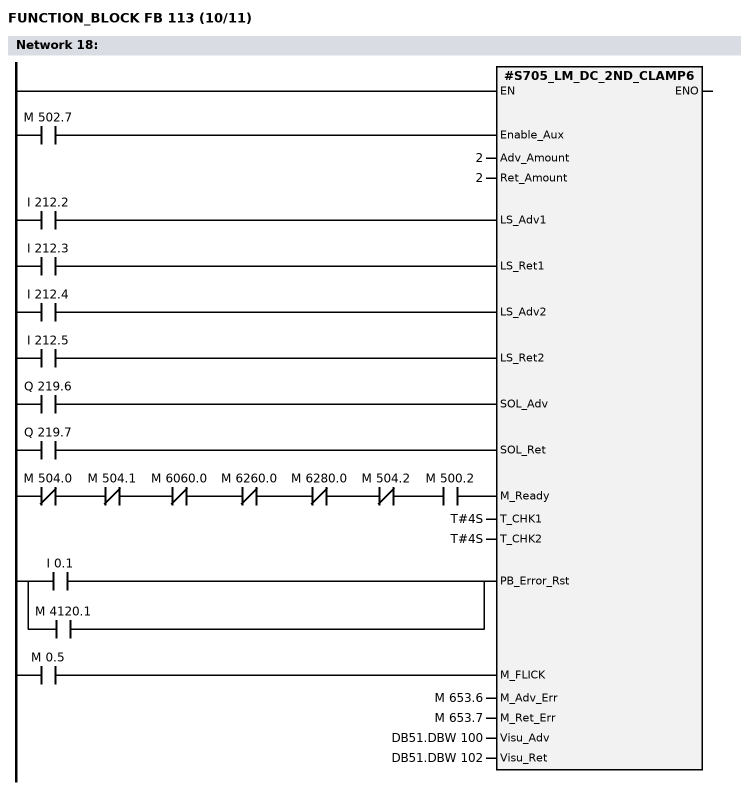

      A     M    502.7;
      =     L      0.0;
      BLD   103;
      A     I    212.2;
      =     L      0.1;
      BLD   103;
      A     I    212.3;
      =     L      0.2;
      BLD   103;
      A     I    212.4;
      =     L      0.3;
      BLD   103;
      A     I    212.5;
      =     L      0.4;
      BLD   103;
      A     Q    219.6;
      =     L      1.1;
      BLD   103;
      A     Q    219.7;
      =     L      1.2;
      BLD   103;
      AN    M    504.0;
      AN    M    504.1;
      AN    M   6060.0;
      AN    M   6260.0;
      AN    M   6280.0;
      AN    M    504.2;
      A     M    500.2;
      =     L      1.3;
      BLD   103;
      A(    ;
      O     I      0.1;
      O     M   4120.1;
      )     ;
      =     L      1.5;
      BLD   103;
      A     M      0.5;
      =     L      1.6;
      BLD   103;
      CALL #S705_LM_DC_2ND_CLAMP6 (
           Enable_Aux               := L      0.0,
           Adv_Amount               := 2,
           Ret_Amount               := 2,
           LS_Adv1                  := L      0.1,
           LS_Ret1                  := L      0.2,
           LS_Adv2                  := L      0.3,
           LS_Ret2                  := L      0.4,
           SOL_Adv                  := L      1.1,
           SOL_Ret                  := L      1.2,
           M_Ready                  := L      1.3,
           T_CHK1                   := T#4S,
           T_CHK2                   := T#4S,
           PB_Error_Rst             := L      1.5,
           M_FLICK                  := L      1.6,
           M_Adv_Err                := M    653.6,
           M_Ret_Err                := M    653.7,
           Visu_Adv                 := DB51.DBW  100,
           Visu_Ret                 := DB51.DBW  102);
      NOP   0;
NETWORK
TITLE =
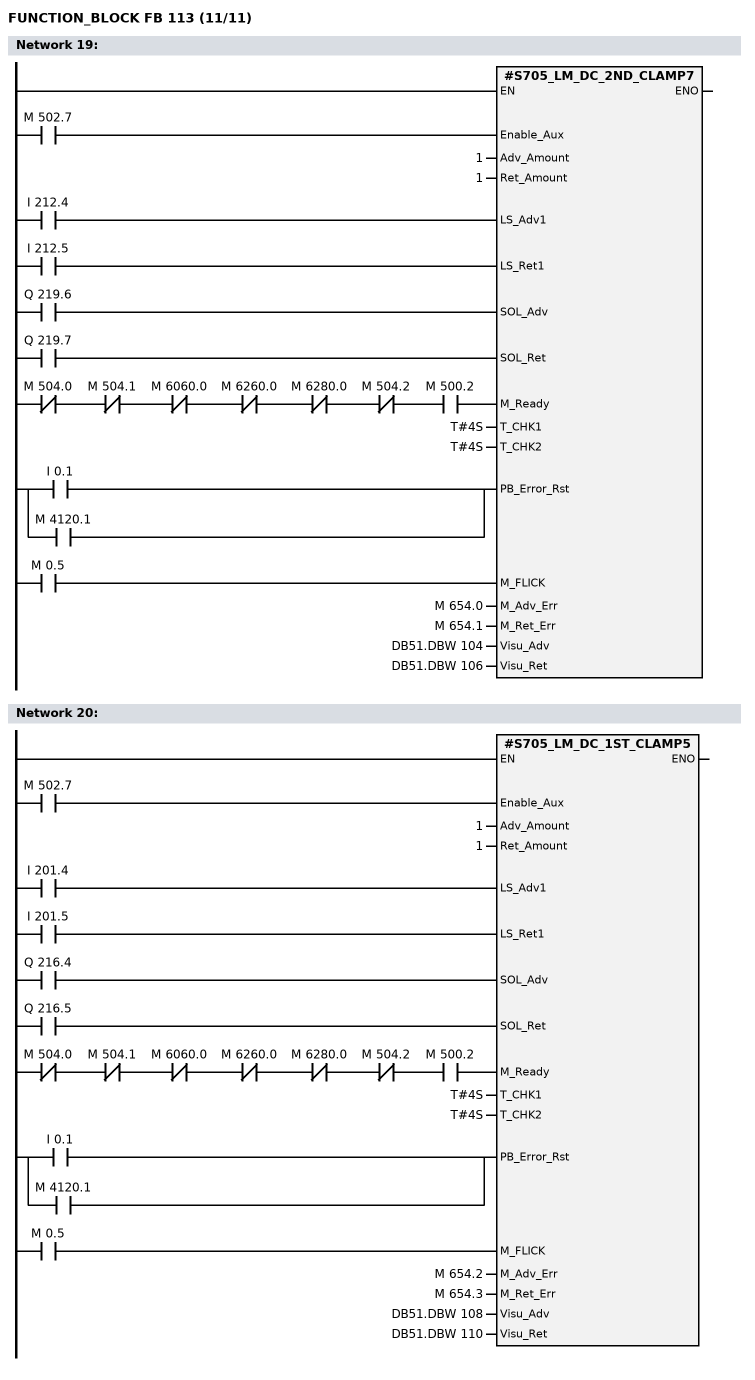

      A     M    502.7;
      =     L      0.0;
      BLD   103;
      A     I    212.4;
      =     L      0.1;
      BLD   103;
      A     I    212.5;
      =     L      0.2;
      BLD   103;
      A     Q    219.6;
      =     L      1.1;
      BLD   103;
      A     Q    219.7;
      =     L      1.2;
      BLD   103;
      AN    M    504.0;
      AN    M    504.1;
      AN    M   6060.0;
      AN    M   6260.0;
      AN    M   6280.0;
      AN    M    504.2;
      A     M    500.2;
      =     L      1.3;
      BLD   103;
      A(    ;
      O     I      0.1;
      O     M   4120.1;
      )     ;
      =     L      1.5;
      BLD   103;
      A     M      0.5;
      =     L      1.6;
      BLD   103;
      CALL #S705_LM_DC_2ND_CLAMP7 (
           Enable_Aux               := L      0.0,
           Adv_Amount               := 1,
           Ret_Amount               := 1,
           LS_Adv1                  := L      0.1,
           LS_Ret1                  := L      0.2,
           SOL_Adv                  := L      1.1,
           SOL_Ret                  := L      1.2,
           M_Ready                  := L      1.3,
           T_CHK1                   := T#4S,
           T_CHK2                   := T#4S,
           PB_Error_Rst             := L      1.5,
           M_FLICK                  := L      1.6,
           M_Adv_Err                := M    654.0,
           M_Ret_Err                := M    654.1,
           Visu_Adv                 := DB51.DBW  104,
           Visu_Ret                 := DB51.DBW  106);
      NOP   0;
NETWORK
TITLE =

      A     M    502.7;
      =     L      0.0;
      BLD   103;
      A     I    201.4;
      =     L      0.1;
      BLD   103;
      A     I    201.5;
      =     L      0.2;
      BLD   103;
      A     Q    216.4;
      =     L      1.1;
      BLD   103;
      A     Q    216.5;
      =     L      1.2;
      BLD   103;
      AN    M    504.0;
      AN    M    504.1;
      AN    M   6060.0;
      AN    M   6260.0;
      AN    M   6280.0;
      AN    M    504.2;
      A     M    500.2;
      =     L      1.3;
      BLD   103;
      A(    ;
      O     I      0.1;
      O     M   4120.1;
      )     ;
      =     L      1.5;
      BLD   103;
      A     M      0.5;
      =     L      1.6;
      BLD   103;
      CALL #S705_LM_DC_1ST_CLAMP5 (
           Enable_Aux               := L      0.0,
           Adv_Amount               := 1,
           Ret_Amount               := 1,
           LS_Adv1                  := L      0.1,
           LS_Ret1                  := L      0.2,
           SOL_Adv                  := L      1.1,
           SOL_Ret                  := L      1.2,
           M_Ready                  := L      1.3,
           T_CHK1                   := T#4S,
           T_CHK2                   := T#4S,
           PB_Error_Rst             := L      1.5,
           M_FLICK                  := L      1.6,
           M_Adv_Err                := M    654.2,
           M_Ret_Err                := M    654.3,
           Visu_Adv                 := DB51.DBW  108,
           Visu_Ret                 := DB51.DBW  110);
      NOP   0;
END_FUNCTION_BLOCK

DATA_BLOCK DB 113
TITLE =
VERSION : 0.0

 FB 113
BEGIN
   S705_LM_DC_PIN.Enable_Aux := FALSE;
   S705_LM_DC_PIN.Adv_Amount := 1;
   S705_LM_DC_PIN.Ret_Amount := 1;
   S705_LM_DC_PIN.LS_Adv1 := FALSE;
   S705_LM_DC_PIN.LS_Ret1 := FALSE;
   S705_LM_DC_PIN.LS_Adv2 := FALSE;
   S705_LM_DC_PIN.LS_Ret2 := FALSE;
   S705_LM_DC_PIN.LS_Adv3 := FALSE;
   S705_LM_DC_PIN.LS_Ret3 := FALSE;
   S705_LM_DC_PIN.LS_Adv4 := FALSE;
   S705_LM_DC_PIN.LS_Ret4 := FALSE;
   S705_LM_DC_PIN.SOL_Adv := FALSE;
   S705_LM_DC_PIN.SOL_Ret := FALSE;
   S705_LM_DC_PIN.M_Ready := TRUE;
   S705_LM_DC_PIN.T_CHK1 := T#4S;
   S705_LM_DC_PIN.T_CHK2 := T#4S;
   S705_LM_DC_PIN.PB_Lamp_CHK := FALSE;
   S705_LM_DC_PIN.PB_Error_Rst := FALSE;
   S705_LM_DC_PIN.M_FLICK := TRUE;
   S705_LM_DC_PIN.M_Adv_Err := FALSE;
   S705_LM_DC_PIN.M_Ret_Err := FALSE;
   S705_LM_DC_PIN.LP_Adv := FALSE;
   S705_LM_DC_PIN.LP_Ret := FALSE;
   S705_LM_DC_PIN.Visu_Adv := W#16#0;
   S705_LM_DC_PIN.Visu_Ret := W#16#0;
   S705_LM_DC_PIN.Error_T1.IN := FALSE;
   S705_LM_DC_PIN.Error_T1.PT := T#4S;
   S705_LM_DC_PIN.Error_T1.Q := FALSE;
   S705_LM_DC_PIN.Error_T1.ET := T#0MS;
   S705_LM_DC_PIN.Error_T1.STATE := B#16#0;
   S705_LM_DC_PIN.Error_T1.STIME := T#15D15H9M7S743MS;
   S705_LM_DC_PIN.Error_T1.ATIME := T#15D15H9M7S788MS;
   S705_LM_DC_PIN.Error_T2.IN := FALSE;
   S705_LM_DC_PIN.Error_T2.PT := T#4S;
   S705_LM_DC_PIN.Error_T2.Q := FALSE;
   S705_LM_DC_PIN.Error_T2.ET := T#0MS;
   S705_LM_DC_PIN.Error_T2.STATE := B#16#0;
   S705_LM_DC_PIN.Error_T2.STIME := T#0MS;
   S705_LM_DC_PIN.Error_T2.ATIME := T#0MS;
   S705_LM_DC_PIN.CHK_Aux1 := FALSE;
   S705_LM_DC_PIN.CHK_Aux2 := FALSE;
   S705_LM_DC_PIN.Error_T1_DN := FALSE;
   S705_LM_DC_PIN.Error_T2_DN := FALSE;
   S705_LM_DC_PIN.Adv_Memo := TRUE;
   S705_LM_DC_PIN.Visu_Adv_Arr[0] := FALSE;
   S705_LM_DC_PIN.Visu_Adv_Arr[1] := FALSE;
   S705_LM_DC_PIN.Visu_Adv_Arr[2] := FALSE;
   S705_LM_DC_PIN.Visu_Adv_Arr[3] := FALSE;
   S705_LM_DC_PIN.Visu_Adv_Arr[4] := FALSE;
   S705_LM_DC_PIN.Visu_Adv_Arr[5] := FALSE;
   S705_LM_DC_PIN.Visu_Adv_Arr[6] := FALSE;
   S705_LM_DC_PIN.Visu_Adv_Arr[7] := FALSE;
   S705_LM_DC_PIN.Visu_Adv_Arr[8] := FALSE;
   S705_LM_DC_PIN.Visu_Adv_Arr[9] := FALSE;
   S705_LM_DC_PIN.Visu_Adv_Arr[10] := FALSE;
   S705_LM_DC_PIN.Visu_Adv_Arr[11] := FALSE;
   S705_LM_DC_PIN.Visu_Adv_Arr[12] := FALSE;
   S705_LM_DC_PIN.Visu_Adv_Arr[13] := FALSE;
   S705_LM_DC_PIN.Visu_Adv_Arr[14] := FALSE;
   S705_LM_DC_PIN.Visu_Adv_Arr[15] := FALSE;
   S705_LM_DC_PIN.Visu_Ret_Arr[0] := FALSE;
   S705_LM_DC_PIN.Visu_Ret_Arr[1] := FALSE;
   S705_LM_DC_PIN.Visu_Ret_Arr[2] := FALSE;
   S705_LM_DC_PIN.Visu_Ret_Arr[3] := FALSE;
   S705_LM_DC_PIN.Visu_Ret_Arr[4] := FALSE;
   S705_LM_DC_PIN.Visu_Ret_Arr[5] := FALSE;
   S705_LM_DC_PIN.Visu_Ret_Arr[6] := FALSE;
   S705_LM_DC_PIN.Visu_Ret_Arr[7] := FALSE;
   S705_LM_DC_PIN.Visu_Ret_Arr[8] := FALSE;
   S705_LM_DC_PIN.Visu_Ret_Arr[9] := FALSE;
   S705_LM_DC_PIN.Visu_Ret_Arr[10] := FALSE;
   S705_LM_DC_PIN.Visu_Ret_Arr[11] := FALSE;
   S705_LM_DC_PIN.Visu_Ret_Arr[12] := FALSE;
   S705_LM_DC_PIN.Visu_Ret_Arr[13] := FALSE;
   S705_LM_DC_PIN.Visu_Ret_Arr[14] := FALSE;
   S705_LM_DC_PIN.Visu_Ret_Arr[15] := FALSE;
   S705_LM_DC_PIN.BLK_Move_Ret := 0;
   S705_LM_DC_PIN.Enable := FALSE;
   S705_LM_DC_PIN.Adv_End := FALSE;
   S705_LM_DC_PIN.Ret_End := FALSE;
   S705_LM_DC_1ST_CLAMP1.Enable_Aux := FALSE;
   S705_LM_DC_1ST_CLAMP1.Adv_Amount := 1;
   S705_LM_DC_1ST_CLAMP1.Ret_Amount := 1;
   S705_LM_DC_1ST_CLAMP1.LS_Adv1 := FALSE;
   S705_LM_DC_1ST_CLAMP1.LS_Ret1 := FALSE;
   S705_LM_DC_1ST_CLAMP1.LS_Adv2 := FALSE;
   S705_LM_DC_1ST_CLAMP1.LS_Ret2 := FALSE;
   S705_LM_DC_1ST_CLAMP1.LS_Adv3 := FALSE;
   S705_LM_DC_1ST_CLAMP1.LS_Ret3 := FALSE;
   S705_LM_DC_1ST_CLAMP1.LS_Adv4 := FALSE;
   S705_LM_DC_1ST_CLAMP1.LS_Ret4 := FALSE;
   S705_LM_DC_1ST_CLAMP1.SOL_Adv := FALSE;
   S705_LM_DC_1ST_CLAMP1.SOL_Ret := FALSE;
   S705_LM_DC_1ST_CLAMP1.M_Ready := TRUE;
   S705_LM_DC_1ST_CLAMP1.T_CHK1 := T#4S;
   S705_LM_DC_1ST_CLAMP1.T_CHK2 := T#4S;
   S705_LM_DC_1ST_CLAMP1.PB_Lamp_CHK := FALSE;
   S705_LM_DC_1ST_CLAMP1.PB_Error_Rst := FALSE;
   S705_LM_DC_1ST_CLAMP1.M_FLICK := TRUE;
   S705_LM_DC_1ST_CLAMP1.M_Adv_Err := FALSE;
   S705_LM_DC_1ST_CLAMP1.M_Ret_Err := FALSE;
   S705_LM_DC_1ST_CLAMP1.LP_Adv := FALSE;
   S705_LM_DC_1ST_CLAMP1.LP_Ret := FALSE;
   S705_LM_DC_1ST_CLAMP1.Visu_Adv := W#16#0;
   S705_LM_DC_1ST_CLAMP1.Visu_Ret := W#16#0;
   S705_LM_DC_1ST_CLAMP1.Error_T1.IN := FALSE;
   S705_LM_DC_1ST_CLAMP1.Error_T1.PT := T#4S;
   S705_LM_DC_1ST_CLAMP1.Error_T1.Q := FALSE;
   S705_LM_DC_1ST_CLAMP1.Error_T1.ET := T#0MS;
   S705_LM_DC_1ST_CLAMP1.Error_T1.STATE := B#16#0;
   S705_LM_DC_1ST_CLAMP1.Error_T1.STIME := T#15D15H9M7S743MS;
   S705_LM_DC_1ST_CLAMP1.Error_T1.ATIME := T#15D15H9M7S788MS;
   S705_LM_DC_1ST_CLAMP1.Error_T2.IN := FALSE;
   S705_LM_DC_1ST_CLAMP1.Error_T2.PT := T#4S;
   S705_LM_DC_1ST_CLAMP1.Error_T2.Q := FALSE;
   S705_LM_DC_1ST_CLAMP1.Error_T2.ET := T#0MS;
   S705_LM_DC_1ST_CLAMP1.Error_T2.STATE := B#16#0;
   S705_LM_DC_1ST_CLAMP1.Error_T2.STIME := T#0MS;
   S705_LM_DC_1ST_CLAMP1.Error_T2.ATIME := T#0MS;
   S705_LM_DC_1ST_CLAMP1.CHK_Aux1 := FALSE;
   S705_LM_DC_1ST_CLAMP1.CHK_Aux2 := FALSE;
   S705_LM_DC_1ST_CLAMP1.Error_T1_DN := FALSE;
   S705_LM_DC_1ST_CLAMP1.Error_T2_DN := FALSE;
   S705_LM_DC_1ST_CLAMP1.Adv_Memo := TRUE;
   S705_LM_DC_1ST_CLAMP1.Visu_Adv_Arr[0] := FALSE;
   S705_LM_DC_1ST_CLAMP1.Visu_Adv_Arr[1] := FALSE;
   S705_LM_DC_1ST_CLAMP1.Visu_Adv_Arr[2] := FALSE;
   S705_LM_DC_1ST_CLAMP1.Visu_Adv_Arr[3] := FALSE;
   S705_LM_DC_1ST_CLAMP1.Visu_Adv_Arr[4] := FALSE;
   S705_LM_DC_1ST_CLAMP1.Visu_Adv_Arr[5] := FALSE;
   S705_LM_DC_1ST_CLAMP1.Visu_Adv_Arr[6] := FALSE;
   S705_LM_DC_1ST_CLAMP1.Visu_Adv_Arr[7] := FALSE;
   S705_LM_DC_1ST_CLAMP1.Visu_Adv_Arr[8] := FALSE;
   S705_LM_DC_1ST_CLAMP1.Visu_Adv_Arr[9] := FALSE;
   S705_LM_DC_1ST_CLAMP1.Visu_Adv_Arr[10] := FALSE;
   S705_LM_DC_1ST_CLAMP1.Visu_Adv_Arr[11] := FALSE;
   S705_LM_DC_1ST_CLAMP1.Visu_Adv_Arr[12] := FALSE;
   S705_LM_DC_1ST_CLAMP1.Visu_Adv_Arr[13] := FALSE;
   S705_LM_DC_1ST_CLAMP1.Visu_Adv_Arr[14] := FALSE;
   S705_LM_DC_1ST_CLAMP1.Visu_Adv_Arr[15] := FALSE;
   S705_LM_DC_1ST_CLAMP1.Visu_Ret_Arr[0] := FALSE;
   S705_LM_DC_1ST_CLAMP1.Visu_Ret_Arr[1] := FALSE;
   S705_LM_DC_1ST_CLAMP1.Visu_Ret_Arr[2] := FALSE;
   S705_LM_DC_1ST_CLAMP1.Visu_Ret_Arr[3] := FALSE;
   S705_LM_DC_1ST_CLAMP1.Visu_Ret_Arr[4] := FALSE;
   S705_LM_DC_1ST_CLAMP1.Visu_Ret_Arr[5] := FALSE;
   S705_LM_DC_1ST_CLAMP1.Visu_Ret_Arr[6] := FALSE;
   S705_LM_DC_1ST_CLAMP1.Visu_Ret_Arr[7] := FALSE;
   S705_LM_DC_1ST_CLAMP1.Visu_Ret_Arr[8] := FALSE;
   S705_LM_DC_1ST_CLAMP1.Visu_Ret_Arr[9] := FALSE;
   S705_LM_DC_1ST_CLAMP1.Visu_Ret_Arr[10] := FALSE;
   S705_LM_DC_1ST_CLAMP1.Visu_Ret_Arr[11] := FALSE;
   S705_LM_DC_1ST_CLAMP1.Visu_Ret_Arr[12] := FALSE;
   S705_LM_DC_1ST_CLAMP1.Visu_Ret_Arr[13] := FALSE;
   S705_LM_DC_1ST_CLAMP1.Visu_Ret_Arr[14] := FALSE;
   S705_LM_DC_1ST_CLAMP1.Visu_Ret_Arr[15] := FALSE;
   S705_LM_DC_1ST_CLAMP1.BLK_Move_Ret := 0;
   S705_LM_DC_1ST_CLAMP1.Enable := FALSE;
   S705_LM_DC_1ST_CLAMP1.Adv_End := FALSE;
   S705_LM_DC_1ST_CLAMP1.Ret_End := FALSE;
   S705_LM_DC_1ST_CLAMP2.Enable_Aux := FALSE;
   S705_LM_DC_1ST_CLAMP2.Adv_Amount := 2;
   S705_LM_DC_1ST_CLAMP2.Ret_Amount := 2;
   S705_LM_DC_1ST_CLAMP2.LS_Adv1 := FALSE;
   S705_LM_DC_1ST_CLAMP2.LS_Ret1 := FALSE;
   S705_LM_DC_1ST_CLAMP2.LS_Adv2 := FALSE;
   S705_LM_DC_1ST_CLAMP2.LS_Ret2 := FALSE;
   S705_LM_DC_1ST_CLAMP2.LS_Adv3 := FALSE;
   S705_LM_DC_1ST_CLAMP2.LS_Ret3 := FALSE;
   S705_LM_DC_1ST_CLAMP2.LS_Adv4 := FALSE;
   S705_LM_DC_1ST_CLAMP2.LS_Ret4 := FALSE;
   S705_LM_DC_1ST_CLAMP2.SOL_Adv := FALSE;
   S705_LM_DC_1ST_CLAMP2.SOL_Ret := FALSE;
   S705_LM_DC_1ST_CLAMP2.M_Ready := TRUE;
   S705_LM_DC_1ST_CLAMP2.T_CHK1 := T#4S;
   S705_LM_DC_1ST_CLAMP2.T_CHK2 := T#4S;
   S705_LM_DC_1ST_CLAMP2.PB_Lamp_CHK := FALSE;
   S705_LM_DC_1ST_CLAMP2.PB_Error_Rst := FALSE;
   S705_LM_DC_1ST_CLAMP2.M_FLICK := TRUE;
   S705_LM_DC_1ST_CLAMP2.M_Adv_Err := FALSE;
   S705_LM_DC_1ST_CLAMP2.M_Ret_Err := FALSE;
   S705_LM_DC_1ST_CLAMP2.LP_Adv := FALSE;
   S705_LM_DC_1ST_CLAMP2.LP_Ret := FALSE;
   S705_LM_DC_1ST_CLAMP2.Visu_Adv := W#16#0;
   S705_LM_DC_1ST_CLAMP2.Visu_Ret := W#16#0;
   S705_LM_DC_1ST_CLAMP2.Error_T1.IN := FALSE;
   S705_LM_DC_1ST_CLAMP2.Error_T1.PT := T#4S;
   S705_LM_DC_1ST_CLAMP2.Error_T1.Q := FALSE;
   S705_LM_DC_1ST_CLAMP2.Error_T1.ET := T#0MS;
   S705_LM_DC_1ST_CLAMP2.Error_T1.STATE := B#16#0;
   S705_LM_DC_1ST_CLAMP2.Error_T1.STIME := T#22D22H55M12S68MS;
   S705_LM_DC_1ST_CLAMP2.Error_T1.ATIME := T#22D22H55M12S817MS;
   S705_LM_DC_1ST_CLAMP2.Error_T2.IN := FALSE;
   S705_LM_DC_1ST_CLAMP2.Error_T2.PT := T#4S;
   S705_LM_DC_1ST_CLAMP2.Error_T2.Q := FALSE;
   S705_LM_DC_1ST_CLAMP2.Error_T2.ET := T#0MS;
   S705_LM_DC_1ST_CLAMP2.Error_T2.STATE := B#16#0;
   S705_LM_DC_1ST_CLAMP2.Error_T2.STIME := T#0MS;
   S705_LM_DC_1ST_CLAMP2.Error_T2.ATIME := T#0MS;
   S705_LM_DC_1ST_CLAMP2.CHK_Aux1 := FALSE;
   S705_LM_DC_1ST_CLAMP2.CHK_Aux2 := FALSE;
   S705_LM_DC_1ST_CLAMP2.Error_T1_DN := FALSE;
   S705_LM_DC_1ST_CLAMP2.Error_T2_DN := FALSE;
   S705_LM_DC_1ST_CLAMP2.Adv_Memo := TRUE;
   S705_LM_DC_1ST_CLAMP2.Visu_Adv_Arr[0] := FALSE;
   S705_LM_DC_1ST_CLAMP2.Visu_Adv_Arr[1] := FALSE;
   S705_LM_DC_1ST_CLAMP2.Visu_Adv_Arr[2] := FALSE;
   S705_LM_DC_1ST_CLAMP2.Visu_Adv_Arr[3] := FALSE;
   S705_LM_DC_1ST_CLAMP2.Visu_Adv_Arr[4] := FALSE;
   S705_LM_DC_1ST_CLAMP2.Visu_Adv_Arr[5] := FALSE;
   S705_LM_DC_1ST_CLAMP2.Visu_Adv_Arr[6] := FALSE;
   S705_LM_DC_1ST_CLAMP2.Visu_Adv_Arr[7] := FALSE;
   S705_LM_DC_1ST_CLAMP2.Visu_Adv_Arr[8] := FALSE;
   S705_LM_DC_1ST_CLAMP2.Visu_Adv_Arr[9] := FALSE;
   S705_LM_DC_1ST_CLAMP2.Visu_Adv_Arr[10] := FALSE;
   S705_LM_DC_1ST_CLAMP2.Visu_Adv_Arr[11] := FALSE;
   S705_LM_DC_1ST_CLAMP2.Visu_Adv_Arr[12] := FALSE;
   S705_LM_DC_1ST_CLAMP2.Visu_Adv_Arr[13] := FALSE;
   S705_LM_DC_1ST_CLAMP2.Visu_Adv_Arr[14] := FALSE;
   S705_LM_DC_1ST_CLAMP2.Visu_Adv_Arr[15] := FALSE;
   S705_LM_DC_1ST_CLAMP2.Visu_Ret_Arr[0] := FALSE;
   S705_LM_DC_1ST_CLAMP2.Visu_Ret_Arr[1] := FALSE;
   S705_LM_DC_1ST_CLAMP2.Visu_Ret_Arr[2] := FALSE;
   S705_LM_DC_1ST_CLAMP2.Visu_Ret_Arr[3] := FALSE;
   S705_LM_DC_1ST_CLAMP2.Visu_Ret_Arr[4] := FALSE;
   S705_LM_DC_1ST_CLAMP2.Visu_Ret_Arr[5] := FALSE;
   S705_LM_DC_1ST_CLAMP2.Visu_Ret_Arr[6] := FALSE;
   S705_LM_DC_1ST_CLAMP2.Visu_Ret_Arr[7] := FALSE;
   S705_LM_DC_1ST_CLAMP2.Visu_Ret_Arr[8] := FALSE;
   S705_LM_DC_1ST_CLAMP2.Visu_Ret_Arr[9] := FALSE;
   S705_LM_DC_1ST_CLAMP2.Visu_Ret_Arr[10] := FALSE;
   S705_LM_DC_1ST_CLAMP2.Visu_Ret_Arr[11] := FALSE;
   S705_LM_DC_1ST_CLAMP2.Visu_Ret_Arr[12] := FALSE;
   S705_LM_DC_1ST_CLAMP2.Visu_Ret_Arr[13] := FALSE;
   S705_LM_DC_1ST_CLAMP2.Visu_Ret_Arr[14] := FALSE;
   S705_LM_DC_1ST_CLAMP2.Visu_Ret_Arr[15] := FALSE;
   S705_LM_DC_1ST_CLAMP2.BLK_Move_Ret := 0;
   S705_LM_DC_1ST_CLAMP2.Enable := FALSE;
   S705_LM_DC_1ST_CLAMP2.Adv_End := FALSE;
   S705_LM_DC_1ST_CLAMP2.Ret_End := FALSE;
   S705_LM_DC_1ST_CLAMP3.Enable_Aux := FALSE;
   S705_LM_DC_1ST_CLAMP3.Adv_Amount := 1;
   S705_LM_DC_1ST_CLAMP3.Ret_Amount := 1;
   S705_LM_DC_1ST_CLAMP3.LS_Adv1 := FALSE;
   S705_LM_DC_1ST_CLAMP3.LS_Ret1 := FALSE;
   S705_LM_DC_1ST_CLAMP3.LS_Adv2 := FALSE;
   S705_LM_DC_1ST_CLAMP3.LS_Ret2 := FALSE;
   S705_LM_DC_1ST_CLAMP3.LS_Adv3 := FALSE;
   S705_LM_DC_1ST_CLAMP3.LS_Ret3 := FALSE;
   S705_LM_DC_1ST_CLAMP3.LS_Adv4 := FALSE;
   S705_LM_DC_1ST_CLAMP3.LS_Ret4 := FALSE;
   S705_LM_DC_1ST_CLAMP3.SOL_Adv := FALSE;
   S705_LM_DC_1ST_CLAMP3.SOL_Ret := FALSE;
   S705_LM_DC_1ST_CLAMP3.M_Ready := TRUE;
   S705_LM_DC_1ST_CLAMP3.T_CHK1 := T#4S;
   S705_LM_DC_1ST_CLAMP3.T_CHK2 := T#4S;
   S705_LM_DC_1ST_CLAMP3.PB_Lamp_CHK := FALSE;
   S705_LM_DC_1ST_CLAMP3.PB_Error_Rst := FALSE;
   S705_LM_DC_1ST_CLAMP3.M_FLICK := TRUE;
   S705_LM_DC_1ST_CLAMP3.M_Adv_Err := FALSE;
   S705_LM_DC_1ST_CLAMP3.M_Ret_Err := FALSE;
   S705_LM_DC_1ST_CLAMP3.LP_Adv := FALSE;
   S705_LM_DC_1ST_CLAMP3.LP_Ret := FALSE;
   S705_LM_DC_1ST_CLAMP3.Visu_Adv := W#16#0;
   S705_LM_DC_1ST_CLAMP3.Visu_Ret := W#16#0;
   S705_LM_DC_1ST_CLAMP3.Error_T1.IN := FALSE;
   S705_LM_DC_1ST_CLAMP3.Error_T1.PT := T#4S;
   S705_LM_DC_1ST_CLAMP3.Error_T1.Q := FALSE;
   S705_LM_DC_1ST_CLAMP3.Error_T1.ET := T#0MS;
   S705_LM_DC_1ST_CLAMP3.Error_T1.STATE := B#16#0;
   S705_LM_DC_1ST_CLAMP3.Error_T1.STIME := T#22D22H55M12S68MS;
   S705_LM_DC_1ST_CLAMP3.Error_T1.ATIME := T#22D22H55M12S726MS;
   S705_LM_DC_1ST_CLAMP3.Error_T2.IN := FALSE;
   S705_LM_DC_1ST_CLAMP3.Error_T2.PT := T#4S;
   S705_LM_DC_1ST_CLAMP3.Error_T2.Q := FALSE;
   S705_LM_DC_1ST_CLAMP3.Error_T2.ET := T#0MS;
   S705_LM_DC_1ST_CLAMP3.Error_T2.STATE := B#16#0;
   S705_LM_DC_1ST_CLAMP3.Error_T2.STIME := T#0MS;
   S705_LM_DC_1ST_CLAMP3.Error_T2.ATIME := T#0MS;
   S705_LM_DC_1ST_CLAMP3.CHK_Aux1 := FALSE;
   S705_LM_DC_1ST_CLAMP3.CHK_Aux2 := FALSE;
   S705_LM_DC_1ST_CLAMP3.Error_T1_DN := FALSE;
   S705_LM_DC_1ST_CLAMP3.Error_T2_DN := FALSE;
   S705_LM_DC_1ST_CLAMP3.Adv_Memo := TRUE;
   S705_LM_DC_1ST_CLAMP3.Visu_Adv_Arr[0] := FALSE;
   S705_LM_DC_1ST_CLAMP3.Visu_Adv_Arr[1] := FALSE;
   S705_LM_DC_1ST_CLAMP3.Visu_Adv_Arr[2] := FALSE;
   S705_LM_DC_1ST_CLAMP3.Visu_Adv_Arr[3] := FALSE;
   S705_LM_DC_1ST_CLAMP3.Visu_Adv_Arr[4] := FALSE;
   S705_LM_DC_1ST_CLAMP3.Visu_Adv_Arr[5] := FALSE;
   S705_LM_DC_1ST_CLAMP3.Visu_Adv_Arr[6] := FALSE;
   S705_LM_DC_1ST_CLAMP3.Visu_Adv_Arr[7] := FALSE;
   S705_LM_DC_1ST_CLAMP3.Visu_Adv_Arr[8] := FALSE;
   S705_LM_DC_1ST_CLAMP3.Visu_Adv_Arr[9] := FALSE;
   S705_LM_DC_1ST_CLAMP3.Visu_Adv_Arr[10] := FALSE;
   S705_LM_DC_1ST_CLAMP3.Visu_Adv_Arr[11] := FALSE;
   S705_LM_DC_1ST_CLAMP3.Visu_Adv_Arr[12] := FALSE;
   S705_LM_DC_1ST_CLAMP3.Visu_Adv_Arr[13] := FALSE;
   S705_LM_DC_1ST_CLAMP3.Visu_Adv_Arr[14] := FALSE;
   S705_LM_DC_1ST_CLAMP3.Visu_Adv_Arr[15] := FALSE;
   S705_LM_DC_1ST_CLAMP3.Visu_Ret_Arr[0] := FALSE;
   S705_LM_DC_1ST_CLAMP3.Visu_Ret_Arr[1] := FALSE;
   S705_LM_DC_1ST_CLAMP3.Visu_Ret_Arr[2] := FALSE;
   S705_LM_DC_1ST_CLAMP3.Visu_Ret_Arr[3] := FALSE;
   S705_LM_DC_1ST_CLAMP3.Visu_Ret_Arr[4] := FALSE;
   S705_LM_DC_1ST_CLAMP3.Visu_Ret_Arr[5] := FALSE;
   S705_LM_DC_1ST_CLAMP3.Visu_Ret_Arr[6] := FALSE;
   S705_LM_DC_1ST_CLAMP3.Visu_Ret_Arr[7] := FALSE;
   S705_LM_DC_1ST_CLAMP3.Visu_Ret_Arr[8] := FALSE;
   S705_LM_DC_1ST_CLAMP3.Visu_Ret_Arr[9] := FALSE;
   S705_LM_DC_1ST_CLAMP3.Visu_Ret_Arr[10] := FALSE;
   S705_LM_DC_1ST_CLAMP3.Visu_Ret_Arr[11] := FALSE;
   S705_LM_DC_1ST_CLAMP3.Visu_Ret_Arr[12] := FALSE;
   S705_LM_DC_1ST_CLAMP3.Visu_Ret_Arr[13] := FALSE;
   S705_LM_DC_1ST_CLAMP3.Visu_Ret_Arr[14] := FALSE;
   S705_LM_DC_1ST_CLAMP3.Visu_Ret_Arr[15] := FALSE;
   S705_LM_DC_1ST_CLAMP3.BLK_Move_Ret := 0;
   S705_LM_DC_1ST_CLAMP3.Enable := FALSE;
   S705_LM_DC_1ST_CLAMP3.Adv_End := FALSE;
   S705_LM_DC_1ST_CLAMP3.Ret_End := FALSE;
   S705_LM_DC_1ST_CLAMP4.Enable_Aux := FALSE;
   S705_LM_DC_1ST_CLAMP4.Adv_Amount := 1;
   S705_LM_DC_1ST_CLAMP4.Ret_Amount := 1;
   S705_LM_DC_1ST_CLAMP4.LS_Adv1 := FALSE;
   S705_LM_DC_1ST_CLAMP4.LS_Ret1 := FALSE;
   S705_LM_DC_1ST_CLAMP4.LS_Adv2 := FALSE;
   S705_LM_DC_1ST_CLAMP4.LS_Ret2 := FALSE;
   S705_LM_DC_1ST_CLAMP4.LS_Adv3 := FALSE;
   S705_LM_DC_1ST_CLAMP4.LS_Ret3 := FALSE;
   S705_LM_DC_1ST_CLAMP4.LS_Adv4 := FALSE;
   S705_LM_DC_1ST_CLAMP4.LS_Ret4 := FALSE;
   S705_LM_DC_1ST_CLAMP4.SOL_Adv := FALSE;
   S705_LM_DC_1ST_CLAMP4.SOL_Ret := FALSE;
   S705_LM_DC_1ST_CLAMP4.M_Ready := TRUE;
   S705_LM_DC_1ST_CLAMP4.T_CHK1 := T#4S;
   S705_LM_DC_1ST_CLAMP4.T_CHK2 := T#4S;
   S705_LM_DC_1ST_CLAMP4.PB_Lamp_CHK := FALSE;
   S705_LM_DC_1ST_CLAMP4.PB_Error_Rst := FALSE;
   S705_LM_DC_1ST_CLAMP4.M_FLICK := TRUE;
   S705_LM_DC_1ST_CLAMP4.M_Adv_Err := FALSE;
   S705_LM_DC_1ST_CLAMP4.M_Ret_Err := FALSE;
   S705_LM_DC_1ST_CLAMP4.LP_Adv := FALSE;
   S705_LM_DC_1ST_CLAMP4.LP_Ret := FALSE;
   S705_LM_DC_1ST_CLAMP4.Visu_Adv := W#16#0;
   S705_LM_DC_1ST_CLAMP4.Visu_Ret := W#16#0;
   S705_LM_DC_1ST_CLAMP4.Error_T1.IN := FALSE;
   S705_LM_DC_1ST_CLAMP4.Error_T1.PT := T#4S;
   S705_LM_DC_1ST_CLAMP4.Error_T1.Q := FALSE;
   S705_LM_DC_1ST_CLAMP4.Error_T1.ET := T#0MS;
   S705_LM_DC_1ST_CLAMP4.Error_T1.STATE := B#16#0;
   S705_LM_DC_1ST_CLAMP4.Error_T1.STIME := T#22D22H55M13S;
   S705_LM_DC_1ST_CLAMP4.Error_T1.ATIME := T#22D22H55M13S46MS;
   S705_LM_DC_1ST_CLAMP4.Error_T2.IN := FALSE;
   S705_LM_DC_1ST_CLAMP4.Error_T2.PT := T#4S;
   S705_LM_DC_1ST_CLAMP4.Error_T2.Q := FALSE;
   S705_LM_DC_1ST_CLAMP4.Error_T2.ET := T#0MS;
   S705_LM_DC_1ST_CLAMP4.Error_T2.STATE := B#16#0;
   S705_LM_DC_1ST_CLAMP4.Error_T2.STIME := T#0MS;
   S705_LM_DC_1ST_CLAMP4.Error_T2.ATIME := T#0MS;
   S705_LM_DC_1ST_CLAMP4.CHK_Aux1 := FALSE;
   S705_LM_DC_1ST_CLAMP4.CHK_Aux2 := FALSE;
   S705_LM_DC_1ST_CLAMP4.Error_T1_DN := FALSE;
   S705_LM_DC_1ST_CLAMP4.Error_T2_DN := FALSE;
   S705_LM_DC_1ST_CLAMP4.Adv_Memo := TRUE;
   S705_LM_DC_1ST_CLAMP4.Visu_Adv_Arr[0] := FALSE;
   S705_LM_DC_1ST_CLAMP4.Visu_Adv_Arr[1] := FALSE;
   S705_LM_DC_1ST_CLAMP4.Visu_Adv_Arr[2] := FALSE;
   S705_LM_DC_1ST_CLAMP4.Visu_Adv_Arr[3] := FALSE;
   S705_LM_DC_1ST_CLAMP4.Visu_Adv_Arr[4] := FALSE;
   S705_LM_DC_1ST_CLAMP4.Visu_Adv_Arr[5] := FALSE;
   S705_LM_DC_1ST_CLAMP4.Visu_Adv_Arr[6] := FALSE;
   S705_LM_DC_1ST_CLAMP4.Visu_Adv_Arr[7] := FALSE;
   S705_LM_DC_1ST_CLAMP4.Visu_Adv_Arr[8] := FALSE;
   S705_LM_DC_1ST_CLAMP4.Visu_Adv_Arr[9] := FALSE;
   S705_LM_DC_1ST_CLAMP4.Visu_Adv_Arr[10] := FALSE;
   S705_LM_DC_1ST_CLAMP4.Visu_Adv_Arr[11] := FALSE;
   S705_LM_DC_1ST_CLAMP4.Visu_Adv_Arr[12] := FALSE;
   S705_LM_DC_1ST_CLAMP4.Visu_Adv_Arr[13] := FALSE;
   S705_LM_DC_1ST_CLAMP4.Visu_Adv_Arr[14] := FALSE;
   S705_LM_DC_1ST_CLAMP4.Visu_Adv_Arr[15] := FALSE;
   S705_LM_DC_1ST_CLAMP4.Visu_Ret_Arr[0] := FALSE;
   S705_LM_DC_1ST_CLAMP4.Visu_Ret_Arr[1] := FALSE;
   S705_LM_DC_1ST_CLAMP4.Visu_Ret_Arr[2] := FALSE;
   S705_LM_DC_1ST_CLAMP4.Visu_Ret_Arr[3] := FALSE;
   S705_LM_DC_1ST_CLAMP4.Visu_Ret_Arr[4] := FALSE;
   S705_LM_DC_1ST_CLAMP4.Visu_Ret_Arr[5] := FALSE;
   S705_LM_DC_1ST_CLAMP4.Visu_Ret_Arr[6] := FALSE;
   S705_LM_DC_1ST_CLAMP4.Visu_Ret_Arr[7] := FALSE;
   S705_LM_DC_1ST_CLAMP4.Visu_Ret_Arr[8] := FALSE;
   S705_LM_DC_1ST_CLAMP4.Visu_Ret_Arr[9] := FALSE;
   S705_LM_DC_1ST_CLAMP4.Visu_Ret_Arr[10] := FALSE;
   S705_LM_DC_1ST_CLAMP4.Visu_Ret_Arr[11] := FALSE;
   S705_LM_DC_1ST_CLAMP4.Visu_Ret_Arr[12] := FALSE;
   S705_LM_DC_1ST_CLAMP4.Visu_Ret_Arr[13] := FALSE;
   S705_LM_DC_1ST_CLAMP4.Visu_Ret_Arr[14] := FALSE;
   S705_LM_DC_1ST_CLAMP4.Visu_Ret_Arr[15] := FALSE;
   S705_LM_DC_1ST_CLAMP4.BLK_Move_Ret := 0;
   S705_LM_DC_1ST_CLAMP4.Enable := FALSE;
   S705_LM_DC_1ST_CLAMP4.Adv_End := FALSE;
   S705_LM_DC_1ST_CLAMP4.Ret_End := FALSE;
   S705_LM_DC_2ND_CLAMP1.Enable_Aux := FALSE;
   S705_LM_DC_2ND_CLAMP1.Adv_Amount := 2;
   S705_LM_DC_2ND_CLAMP1.Ret_Amount := 1;
   S705_LM_DC_2ND_CLAMP1.LS_Adv1 := FALSE;
   S705_LM_DC_2ND_CLAMP1.LS_Ret1 := FALSE;
   S705_LM_DC_2ND_CLAMP1.LS_Adv2 := FALSE;
   S705_LM_DC_2ND_CLAMP1.LS_Ret2 := FALSE;
   S705_LM_DC_2ND_CLAMP1.LS_Adv3 := FALSE;
   S705_LM_DC_2ND_CLAMP1.LS_Ret3 := FALSE;
   S705_LM_DC_2ND_CLAMP1.LS_Adv4 := FALSE;
   S705_LM_DC_2ND_CLAMP1.LS_Ret4 := FALSE;
   S705_LM_DC_2ND_CLAMP1.SOL_Adv := FALSE;
   S705_LM_DC_2ND_CLAMP1.SOL_Ret := FALSE;
   S705_LM_DC_2ND_CLAMP1.M_Ready := TRUE;
   S705_LM_DC_2ND_CLAMP1.T_CHK1 := T#4S;
   S705_LM_DC_2ND_CLAMP1.T_CHK2 := T#4S;
   S705_LM_DC_2ND_CLAMP1.PB_Lamp_CHK := FALSE;
   S705_LM_DC_2ND_CLAMP1.PB_Error_Rst := FALSE;
   S705_LM_DC_2ND_CLAMP1.M_FLICK := TRUE;
   S705_LM_DC_2ND_CLAMP1.M_Adv_Err := FALSE;
   S705_LM_DC_2ND_CLAMP1.M_Ret_Err := FALSE;
   S705_LM_DC_2ND_CLAMP1.LP_Adv := FALSE;
   S705_LM_DC_2ND_CLAMP1.LP_Ret := FALSE;
   S705_LM_DC_2ND_CLAMP1.Visu_Adv := W#16#0;
   S705_LM_DC_2ND_CLAMP1.Visu_Ret := W#16#0;
   S705_LM_DC_2ND_CLAMP1.Error_T1.IN := FALSE;
   S705_LM_DC_2ND_CLAMP1.Error_T1.PT := T#4S;
   S705_LM_DC_2ND_CLAMP1.Error_T1.Q := FALSE;
   S705_LM_DC_2ND_CLAMP1.Error_T1.ET := T#0MS;
   S705_LM_DC_2ND_CLAMP1.Error_T1.STATE := B#16#0;
   S705_LM_DC_2ND_CLAMP1.Error_T1.STIME := T#22D22H55M35S537MS;
   S705_LM_DC_2ND_CLAMP1.Error_T1.ATIME := T#22D22H55M36S828MS;
   S705_LM_DC_2ND_CLAMP1.Error_T2.IN := FALSE;
   S705_LM_DC_2ND_CLAMP1.Error_T2.PT := T#4S;
   S705_LM_DC_2ND_CLAMP1.Error_T2.Q := FALSE;
   S705_LM_DC_2ND_CLAMP1.Error_T2.ET := T#0MS;
   S705_LM_DC_2ND_CLAMP1.Error_T2.STATE := B#16#0;
   S705_LM_DC_2ND_CLAMP1.Error_T2.STIME := T#0MS;
   S705_LM_DC_2ND_CLAMP1.Error_T2.ATIME := T#0MS;
   S705_LM_DC_2ND_CLAMP1.CHK_Aux1 := FALSE;
   S705_LM_DC_2ND_CLAMP1.CHK_Aux2 := FALSE;
   S705_LM_DC_2ND_CLAMP1.Error_T1_DN := FALSE;
   S705_LM_DC_2ND_CLAMP1.Error_T2_DN := FALSE;
   S705_LM_DC_2ND_CLAMP1.Adv_Memo := TRUE;
   S705_LM_DC_2ND_CLAMP1.Visu_Adv_Arr[0] := FALSE;
   S705_LM_DC_2ND_CLAMP1.Visu_Adv_Arr[1] := FALSE;
   S705_LM_DC_2ND_CLAMP1.Visu_Adv_Arr[2] := FALSE;
   S705_LM_DC_2ND_CLAMP1.Visu_Adv_Arr[3] := FALSE;
   S705_LM_DC_2ND_CLAMP1.Visu_Adv_Arr[4] := FALSE;
   S705_LM_DC_2ND_CLAMP1.Visu_Adv_Arr[5] := FALSE;
   S705_LM_DC_2ND_CLAMP1.Visu_Adv_Arr[6] := FALSE;
   S705_LM_DC_2ND_CLAMP1.Visu_Adv_Arr[7] := FALSE;
   S705_LM_DC_2ND_CLAMP1.Visu_Adv_Arr[8] := FALSE;
   S705_LM_DC_2ND_CLAMP1.Visu_Adv_Arr[9] := FALSE;
   S705_LM_DC_2ND_CLAMP1.Visu_Adv_Arr[10] := FALSE;
   S705_LM_DC_2ND_CLAMP1.Visu_Adv_Arr[11] := FALSE;
   S705_LM_DC_2ND_CLAMP1.Visu_Adv_Arr[12] := FALSE;
   S705_LM_DC_2ND_CLAMP1.Visu_Adv_Arr[13] := FALSE;
   S705_LM_DC_2ND_CLAMP1.Visu_Adv_Arr[14] := FALSE;
   S705_LM_DC_2ND_CLAMP1.Visu_Adv_Arr[15] := FALSE;
   S705_LM_DC_2ND_CLAMP1.Visu_Ret_Arr[0] := FALSE;
   S705_LM_DC_2ND_CLAMP1.Visu_Ret_Arr[1] := FALSE;
   S705_LM_DC_2ND_CLAMP1.Visu_Ret_Arr[2] := FALSE;
   S705_LM_DC_2ND_CLAMP1.Visu_Ret_Arr[3] := FALSE;
   S705_LM_DC_2ND_CLAMP1.Visu_Ret_Arr[4] := FALSE;
   S705_LM_DC_2ND_CLAMP1.Visu_Ret_Arr[5] := FALSE;
   S705_LM_DC_2ND_CLAMP1.Visu_Ret_Arr[6] := FALSE;
   S705_LM_DC_2ND_CLAMP1.Visu_Ret_Arr[7] := FALSE;
   S705_LM_DC_2ND_CLAMP1.Visu_Ret_Arr[8] := FALSE;
   S705_LM_DC_2ND_CLAMP1.Visu_Ret_Arr[9] := FALSE;
   S705_LM_DC_2ND_CLAMP1.Visu_Ret_Arr[10] := FALSE;
   S705_LM_DC_2ND_CLAMP1.Visu_Ret_Arr[11] := FALSE;
   S705_LM_DC_2ND_CLAMP1.Visu_Ret_Arr[12] := FALSE;
   S705_LM_DC_2ND_CLAMP1.Visu_Ret_Arr[13] := FALSE;
   S705_LM_DC_2ND_CLAMP1.Visu_Ret_Arr[14] := FALSE;
   S705_LM_DC_2ND_CLAMP1.Visu_Ret_Arr[15] := FALSE;
   S705_LM_DC_2ND_CLAMP1.BLK_Move_Ret := 0;
   S705_LM_DC_2ND_CLAMP1.Enable := FALSE;
   S705_LM_DC_2ND_CLAMP1.Adv_End := FALSE;
   S705_LM_DC_2ND_CLAMP1.Ret_End := FALSE;
   S705_LM_DC_2ND_CLAMP2.Enable_Aux := FALSE;
   S705_LM_DC_2ND_CLAMP2.Adv_Amount := 1;
   S705_LM_DC_2ND_CLAMP2.Ret_Amount := 1;
   S705_LM_DC_2ND_CLAMP2.LS_Adv1 := FALSE;
   S705_LM_DC_2ND_CLAMP2.LS_Ret1 := FALSE;
   S705_LM_DC_2ND_CLAMP2.LS_Adv2 := FALSE;
   S705_LM_DC_2ND_CLAMP2.LS_Ret2 := FALSE;
   S705_LM_DC_2ND_CLAMP2.LS_Adv3 := FALSE;
   S705_LM_DC_2ND_CLAMP2.LS_Ret3 := FALSE;
   S705_LM_DC_2ND_CLAMP2.LS_Adv4 := FALSE;
   S705_LM_DC_2ND_CLAMP2.LS_Ret4 := FALSE;
   S705_LM_DC_2ND_CLAMP2.SOL_Adv := FALSE;
   S705_LM_DC_2ND_CLAMP2.SOL_Ret := FALSE;
   S705_LM_DC_2ND_CLAMP2.M_Ready := TRUE;
   S705_LM_DC_2ND_CLAMP2.T_CHK1 := T#4S;
   S705_LM_DC_2ND_CLAMP2.T_CHK2 := T#4S;
   S705_LM_DC_2ND_CLAMP2.PB_Lamp_CHK := FALSE;
   S705_LM_DC_2ND_CLAMP2.PB_Error_Rst := FALSE;
   S705_LM_DC_2ND_CLAMP2.M_FLICK := TRUE;
   S705_LM_DC_2ND_CLAMP2.M_Adv_Err := FALSE;
   S705_LM_DC_2ND_CLAMP2.M_Ret_Err := FALSE;
   S705_LM_DC_2ND_CLAMP2.LP_Adv := FALSE;
   S705_LM_DC_2ND_CLAMP2.LP_Ret := FALSE;
   S705_LM_DC_2ND_CLAMP2.Visu_Adv := W#16#0;
   S705_LM_DC_2ND_CLAMP2.Visu_Ret := W#16#0;
   S705_LM_DC_2ND_CLAMP2.Error_T1.IN := FALSE;
   S705_LM_DC_2ND_CLAMP2.Error_T1.PT := T#4S;
   S705_LM_DC_2ND_CLAMP2.Error_T1.Q := FALSE;
   S705_LM_DC_2ND_CLAMP2.Error_T1.ET := T#0MS;
   S705_LM_DC_2ND_CLAMP2.Error_T1.STATE := B#16#0;
   S705_LM_DC_2ND_CLAMP2.Error_T1.STIME := T#22D22H55M12S68MS;
   S705_LM_DC_2ND_CLAMP2.Error_T1.ATIME := T#22D22H55M13S364MS;
   S705_LM_DC_2ND_CLAMP2.Error_T2.IN := FALSE;
   S705_LM_DC_2ND_CLAMP2.Error_T2.PT := T#4S;
   S705_LM_DC_2ND_CLAMP2.Error_T2.Q := FALSE;
   S705_LM_DC_2ND_CLAMP2.Error_T2.ET := T#0MS;
   S705_LM_DC_2ND_CLAMP2.Error_T2.STATE := B#16#0;
   S705_LM_DC_2ND_CLAMP2.Error_T2.STIME := T#0MS;
   S705_LM_DC_2ND_CLAMP2.Error_T2.ATIME := T#0MS;
   S705_LM_DC_2ND_CLAMP2.CHK_Aux1 := FALSE;
   S705_LM_DC_2ND_CLAMP2.CHK_Aux2 := FALSE;
   S705_LM_DC_2ND_CLAMP2.Error_T1_DN := FALSE;
   S705_LM_DC_2ND_CLAMP2.Error_T2_DN := FALSE;
   S705_LM_DC_2ND_CLAMP2.Adv_Memo := TRUE;
   S705_LM_DC_2ND_CLAMP2.Visu_Adv_Arr[0] := FALSE;
   S705_LM_DC_2ND_CLAMP2.Visu_Adv_Arr[1] := FALSE;
   S705_LM_DC_2ND_CLAMP2.Visu_Adv_Arr[2] := FALSE;
   S705_LM_DC_2ND_CLAMP2.Visu_Adv_Arr[3] := FALSE;
   S705_LM_DC_2ND_CLAMP2.Visu_Adv_Arr[4] := FALSE;
   S705_LM_DC_2ND_CLAMP2.Visu_Adv_Arr[5] := FALSE;
   S705_LM_DC_2ND_CLAMP2.Visu_Adv_Arr[6] := FALSE;
   S705_LM_DC_2ND_CLAMP2.Visu_Adv_Arr[7] := FALSE;
   S705_LM_DC_2ND_CLAMP2.Visu_Adv_Arr[8] := FALSE;
   S705_LM_DC_2ND_CLAMP2.Visu_Adv_Arr[9] := FALSE;
   S705_LM_DC_2ND_CLAMP2.Visu_Adv_Arr[10] := FALSE;
   S705_LM_DC_2ND_CLAMP2.Visu_Adv_Arr[11] := FALSE;
   S705_LM_DC_2ND_CLAMP2.Visu_Adv_Arr[12] := FALSE;
   S705_LM_DC_2ND_CLAMP2.Visu_Adv_Arr[13] := FALSE;
   S705_LM_DC_2ND_CLAMP2.Visu_Adv_Arr[14] := FALSE;
   S705_LM_DC_2ND_CLAMP2.Visu_Adv_Arr[15] := FALSE;
   S705_LM_DC_2ND_CLAMP2.Visu_Ret_Arr[0] := FALSE;
   S705_LM_DC_2ND_CLAMP2.Visu_Ret_Arr[1] := FALSE;
   S705_LM_DC_2ND_CLAMP2.Visu_Ret_Arr[2] := FALSE;
   S705_LM_DC_2ND_CLAMP2.Visu_Ret_Arr[3] := FALSE;
   S705_LM_DC_2ND_CLAMP2.Visu_Ret_Arr[4] := FALSE;
   S705_LM_DC_2ND_CLAMP2.Visu_Ret_Arr[5] := FALSE;
   S705_LM_DC_2ND_CLAMP2.Visu_Ret_Arr[6] := FALSE;
   S705_LM_DC_2ND_CLAMP2.Visu_Ret_Arr[7] := FALSE;
   S705_LM_DC_2ND_CLAMP2.Visu_Ret_Arr[8] := FALSE;
   S705_LM_DC_2ND_CLAMP2.Visu_Ret_Arr[9] := FALSE;
   S705_LM_DC_2ND_CLAMP2.Visu_Ret_Arr[10] := FALSE;
   S705_LM_DC_2ND_CLAMP2.Visu_Ret_Arr[11] := FALSE;
   S705_LM_DC_2ND_CLAMP2.Visu_Ret_Arr[12] := FALSE;
   S705_LM_DC_2ND_CLAMP2.Visu_Ret_Arr[13] := FALSE;
   S705_LM_DC_2ND_CLAMP2.Visu_Ret_Arr[14] := FALSE;
   S705_LM_DC_2ND_CLAMP2.Visu_Ret_Arr[15] := FALSE;
   S705_LM_DC_2ND_CLAMP2.BLK_Move_Ret := 0;
   S705_LM_DC_2ND_CLAMP2.Enable := FALSE;
   S705_LM_DC_2ND_CLAMP2.Adv_End := FALSE;
   S705_LM_DC_2ND_CLAMP2.Ret_End := FALSE;
   S705_LM_DC_2ND_CLAMP3.Enable_Aux := FALSE;
   S705_LM_DC_2ND_CLAMP3.Adv_Amount := 1;
   S705_LM_DC_2ND_CLAMP3.Ret_Amount := 1;
   S705_LM_DC_2ND_CLAMP3.LS_Adv1 := FALSE;
   S705_LM_DC_2ND_CLAMP3.LS_Ret1 := FALSE;
   S705_LM_DC_2ND_CLAMP3.LS_Adv2 := FALSE;
   S705_LM_DC_2ND_CLAMP3.LS_Ret2 := FALSE;
   S705_LM_DC_2ND_CLAMP3.LS_Adv3 := FALSE;
   S705_LM_DC_2ND_CLAMP3.LS_Ret3 := FALSE;
   S705_LM_DC_2ND_CLAMP3.LS_Adv4 := FALSE;
   S705_LM_DC_2ND_CLAMP3.LS_Ret4 := FALSE;
   S705_LM_DC_2ND_CLAMP3.SOL_Adv := FALSE;
   S705_LM_DC_2ND_CLAMP3.SOL_Ret := FALSE;
   S705_LM_DC_2ND_CLAMP3.M_Ready := TRUE;
   S705_LM_DC_2ND_CLAMP3.T_CHK1 := T#4S;
   S705_LM_DC_2ND_CLAMP3.T_CHK2 := T#4S;
   S705_LM_DC_2ND_CLAMP3.PB_Lamp_CHK := FALSE;
   S705_LM_DC_2ND_CLAMP3.PB_Error_Rst := FALSE;
   S705_LM_DC_2ND_CLAMP3.M_FLICK := TRUE;
   S705_LM_DC_2ND_CLAMP3.M_Adv_Err := FALSE;
   S705_LM_DC_2ND_CLAMP3.M_Ret_Err := FALSE;
   S705_LM_DC_2ND_CLAMP3.LP_Adv := FALSE;
   S705_LM_DC_2ND_CLAMP3.LP_Ret := FALSE;
   S705_LM_DC_2ND_CLAMP3.Visu_Adv := W#16#0;
   S705_LM_DC_2ND_CLAMP3.Visu_Ret := W#16#0;
   S705_LM_DC_2ND_CLAMP3.Error_T1.IN := FALSE;
   S705_LM_DC_2ND_CLAMP3.Error_T1.PT := T#4S;
   S705_LM_DC_2ND_CLAMP3.Error_T1.Q := FALSE;
   S705_LM_DC_2ND_CLAMP3.Error_T1.ET := T#0MS;
   S705_LM_DC_2ND_CLAMP3.Error_T1.STATE := B#16#0;
   S705_LM_DC_2ND_CLAMP3.Error_T1.STIME := T#22D22H55M13S364MS;
   S705_LM_DC_2ND_CLAMP3.Error_T1.ATIME := T#22D22H55M14S182MS;
   S705_LM_DC_2ND_CLAMP3.Error_T2.IN := FALSE;
   S705_LM_DC_2ND_CLAMP3.Error_T2.PT := T#4S;
   S705_LM_DC_2ND_CLAMP3.Error_T2.Q := FALSE;
   S705_LM_DC_2ND_CLAMP3.Error_T2.ET := T#0MS;
   S705_LM_DC_2ND_CLAMP3.Error_T2.STATE := B#16#0;
   S705_LM_DC_2ND_CLAMP3.Error_T2.STIME := T#0MS;
   S705_LM_DC_2ND_CLAMP3.Error_T2.ATIME := T#0MS;
   S705_LM_DC_2ND_CLAMP3.CHK_Aux1 := FALSE;
   S705_LM_DC_2ND_CLAMP3.CHK_Aux2 := FALSE;
   S705_LM_DC_2ND_CLAMP3.Error_T1_DN := FALSE;
   S705_LM_DC_2ND_CLAMP3.Error_T2_DN := FALSE;
   S705_LM_DC_2ND_CLAMP3.Adv_Memo := TRUE;
   S705_LM_DC_2ND_CLAMP3.Visu_Adv_Arr[0] := FALSE;
   S705_LM_DC_2ND_CLAMP3.Visu_Adv_Arr[1] := FALSE;
   S705_LM_DC_2ND_CLAMP3.Visu_Adv_Arr[2] := FALSE;
   S705_LM_DC_2ND_CLAMP3.Visu_Adv_Arr[3] := FALSE;
   S705_LM_DC_2ND_CLAMP3.Visu_Adv_Arr[4] := FALSE;
   S705_LM_DC_2ND_CLAMP3.Visu_Adv_Arr[5] := FALSE;
   S705_LM_DC_2ND_CLAMP3.Visu_Adv_Arr[6] := FALSE;
   S705_LM_DC_2ND_CLAMP3.Visu_Adv_Arr[7] := FALSE;
   S705_LM_DC_2ND_CLAMP3.Visu_Adv_Arr[8] := FALSE;
   S705_LM_DC_2ND_CLAMP3.Visu_Adv_Arr[9] := FALSE;
   S705_LM_DC_2ND_CLAMP3.Visu_Adv_Arr[10] := FALSE;
   S705_LM_DC_2ND_CLAMP3.Visu_Adv_Arr[11] := FALSE;
   S705_LM_DC_2ND_CLAMP3.Visu_Adv_Arr[12] := FALSE;
   S705_LM_DC_2ND_CLAMP3.Visu_Adv_Arr[13] := FALSE;
   S705_LM_DC_2ND_CLAMP3.Visu_Adv_Arr[14] := FALSE;
   S705_LM_DC_2ND_CLAMP3.Visu_Adv_Arr[15] := FALSE;
   S705_LM_DC_2ND_CLAMP3.Visu_Ret_Arr[0] := FALSE;
   S705_LM_DC_2ND_CLAMP3.Visu_Ret_Arr[1] := FALSE;
   S705_LM_DC_2ND_CLAMP3.Visu_Ret_Arr[2] := FALSE;
   S705_LM_DC_2ND_CLAMP3.Visu_Ret_Arr[3] := FALSE;
   S705_LM_DC_2ND_CLAMP3.Visu_Ret_Arr[4] := FALSE;
   S705_LM_DC_2ND_CLAMP3.Visu_Ret_Arr[5] := FALSE;
   S705_LM_DC_2ND_CLAMP3.Visu_Ret_Arr[6] := FALSE;
   S705_LM_DC_2ND_CLAMP3.Visu_Ret_Arr[7] := FALSE;
   S705_LM_DC_2ND_CLAMP3.Visu_Ret_Arr[8] := FALSE;
   S705_LM_DC_2ND_CLAMP3.Visu_Ret_Arr[9] := FALSE;
   S705_LM_DC_2ND_CLAMP3.Visu_Ret_Arr[10] := FALSE;
   S705_LM_DC_2ND_CLAMP3.Visu_Ret_Arr[11] := FALSE;
   S705_LM_DC_2ND_CLAMP3.Visu_Ret_Arr[12] := FALSE;
   S705_LM_DC_2ND_CLAMP3.Visu_Ret_Arr[13] := FALSE;
   S705_LM_DC_2ND_CLAMP3.Visu_Ret_Arr[14] := FALSE;
   S705_LM_DC_2ND_CLAMP3.Visu_Ret_Arr[15] := FALSE;
   S705_LM_DC_2ND_CLAMP3.BLK_Move_Ret := 0;
   S705_LM_DC_2ND_CLAMP3.Enable := FALSE;
   S705_LM_DC_2ND_CLAMP3.Adv_End := FALSE;
   S705_LM_DC_2ND_CLAMP3.Ret_End := FALSE;
   S705_LM_DC_2ND_CLAMP4.Enable_Aux := FALSE;
   S705_LM_DC_2ND_CLAMP4.Adv_Amount := 1;
   S705_LM_DC_2ND_CLAMP4.Ret_Amount := 1;
   S705_LM_DC_2ND_CLAMP4.LS_Adv1 := FALSE;
   S705_LM_DC_2ND_CLAMP4.LS_Ret1 := FALSE;
   S705_LM_DC_2ND_CLAMP4.LS_Adv2 := FALSE;
   S705_LM_DC_2ND_CLAMP4.LS_Ret2 := FALSE;
   S705_LM_DC_2ND_CLAMP4.LS_Adv3 := FALSE;
   S705_LM_DC_2ND_CLAMP4.LS_Ret3 := FALSE;
   S705_LM_DC_2ND_CLAMP4.LS_Adv4 := FALSE;
   S705_LM_DC_2ND_CLAMP4.LS_Ret4 := FALSE;
   S705_LM_DC_2ND_CLAMP4.SOL_Adv := FALSE;
   S705_LM_DC_2ND_CLAMP4.SOL_Ret := FALSE;
   S705_LM_DC_2ND_CLAMP4.M_Ready := TRUE;
   S705_LM_DC_2ND_CLAMP4.T_CHK1 := T#4S;
   S705_LM_DC_2ND_CLAMP4.T_CHK2 := T#4S;
   S705_LM_DC_2ND_CLAMP4.PB_Lamp_CHK := FALSE;
   S705_LM_DC_2ND_CLAMP4.PB_Error_Rst := FALSE;
   S705_LM_DC_2ND_CLAMP4.M_FLICK := TRUE;
   S705_LM_DC_2ND_CLAMP4.M_Adv_Err := FALSE;
   S705_LM_DC_2ND_CLAMP4.M_Ret_Err := FALSE;
   S705_LM_DC_2ND_CLAMP4.LP_Adv := FALSE;
   S705_LM_DC_2ND_CLAMP4.LP_Ret := FALSE;
   S705_LM_DC_2ND_CLAMP4.Visu_Adv := W#16#0;
   S705_LM_DC_2ND_CLAMP4.Visu_Ret := W#16#0;
   S705_LM_DC_2ND_CLAMP4.Error_T1.IN := FALSE;
   S705_LM_DC_2ND_CLAMP4.Error_T1.PT := T#4S;
   S705_LM_DC_2ND_CLAMP4.Error_T1.Q := FALSE;
   S705_LM_DC_2ND_CLAMP4.Error_T1.ET := T#0MS;
   S705_LM_DC_2ND_CLAMP4.Error_T1.STATE := B#16#0;
   S705_LM_DC_2ND_CLAMP4.Error_T1.STIME := T#22D22H55M12S726MS;
   S705_LM_DC_2ND_CLAMP4.Error_T1.ATIME := T#22D22H55M13S364MS;
   S705_LM_DC_2ND_CLAMP4.Error_T2.IN := FALSE;
   S705_LM_DC_2ND_CLAMP4.Error_T2.PT := T#4S;
   S705_LM_DC_2ND_CLAMP4.Error_T2.Q := FALSE;
   S705_LM_DC_2ND_CLAMP4.Error_T2.ET := T#0MS;
   S705_LM_DC_2ND_CLAMP4.Error_T2.STATE := B#16#0;
   S705_LM_DC_2ND_CLAMP4.Error_T2.STIME := T#0MS;
   S705_LM_DC_2ND_CLAMP4.Error_T2.ATIME := T#0MS;
   S705_LM_DC_2ND_CLAMP4.CHK_Aux1 := FALSE;
   S705_LM_DC_2ND_CLAMP4.CHK_Aux2 := FALSE;
   S705_LM_DC_2ND_CLAMP4.Error_T1_DN := FALSE;
   S705_LM_DC_2ND_CLAMP4.Error_T2_DN := FALSE;
   S705_LM_DC_2ND_CLAMP4.Adv_Memo := TRUE;
   S705_LM_DC_2ND_CLAMP4.Visu_Adv_Arr[0] := FALSE;
   S705_LM_DC_2ND_CLAMP4.Visu_Adv_Arr[1] := FALSE;
   S705_LM_DC_2ND_CLAMP4.Visu_Adv_Arr[2] := FALSE;
   S705_LM_DC_2ND_CLAMP4.Visu_Adv_Arr[3] := FALSE;
   S705_LM_DC_2ND_CLAMP4.Visu_Adv_Arr[4] := FALSE;
   S705_LM_DC_2ND_CLAMP4.Visu_Adv_Arr[5] := FALSE;
   S705_LM_DC_2ND_CLAMP4.Visu_Adv_Arr[6] := FALSE;
   S705_LM_DC_2ND_CLAMP4.Visu_Adv_Arr[7] := FALSE;
   S705_LM_DC_2ND_CLAMP4.Visu_Adv_Arr[8] := FALSE;
   S705_LM_DC_2ND_CLAMP4.Visu_Adv_Arr[9] := FALSE;
   S705_LM_DC_2ND_CLAMP4.Visu_Adv_Arr[10] := FALSE;
   S705_LM_DC_2ND_CLAMP4.Visu_Adv_Arr[11] := FALSE;
   S705_LM_DC_2ND_CLAMP4.Visu_Adv_Arr[12] := FALSE;
   S705_LM_DC_2ND_CLAMP4.Visu_Adv_Arr[13] := FALSE;
   S705_LM_DC_2ND_CLAMP4.Visu_Adv_Arr[14] := FALSE;
   S705_LM_DC_2ND_CLAMP4.Visu_Adv_Arr[15] := FALSE;
   S705_LM_DC_2ND_CLAMP4.Visu_Ret_Arr[0] := FALSE;
   S705_LM_DC_2ND_CLAMP4.Visu_Ret_Arr[1] := FALSE;
   S705_LM_DC_2ND_CLAMP4.Visu_Ret_Arr[2] := FALSE;
   S705_LM_DC_2ND_CLAMP4.Visu_Ret_Arr[3] := FALSE;
   S705_LM_DC_2ND_CLAMP4.Visu_Ret_Arr[4] := FALSE;
   S705_LM_DC_2ND_CLAMP4.Visu_Ret_Arr[5] := FALSE;
   S705_LM_DC_2ND_CLAMP4.Visu_Ret_Arr[6] := FALSE;
   S705_LM_DC_2ND_CLAMP4.Visu_Ret_Arr[7] := FALSE;
   S705_LM_DC_2ND_CLAMP4.Visu_Ret_Arr[8] := FALSE;
   S705_LM_DC_2ND_CLAMP4.Visu_Ret_Arr[9] := FALSE;
   S705_LM_DC_2ND_CLAMP4.Visu_Ret_Arr[10] := FALSE;
   S705_LM_DC_2ND_CLAMP4.Visu_Ret_Arr[11] := FALSE;
   S705_LM_DC_2ND_CLAMP4.Visu_Ret_Arr[12] := FALSE;
   S705_LM_DC_2ND_CLAMP4.Visu_Ret_Arr[13] := FALSE;
   S705_LM_DC_2ND_CLAMP4.Visu_Ret_Arr[14] := FALSE;
   S705_LM_DC_2ND_CLAMP4.Visu_Ret_Arr[15] := FALSE;
   S705_LM_DC_2ND_CLAMP4.BLK_Move_Ret := 0;
   S705_LM_DC_2ND_CLAMP4.Enable := FALSE;
   S705_LM_DC_2ND_CLAMP4.Adv_End := FALSE;
   S705_LM_DC_2ND_CLAMP4.Ret_End := FALSE;
   S705_LM_DC_2ND_CLAMP5.Enable_Aux := FALSE;
   S705_LM_DC_2ND_CLAMP5.Adv_Amount := 1;
   S705_LM_DC_2ND_CLAMP5.Ret_Amount := 1;
   S705_LM_DC_2ND_CLAMP5.LS_Adv1 := FALSE;
   S705_LM_DC_2ND_CLAMP5.LS_Ret1 := FALSE;
   S705_LM_DC_2ND_CLAMP5.LS_Adv2 := FALSE;
   S705_LM_DC_2ND_CLAMP5.LS_Ret2 := FALSE;
   S705_LM_DC_2ND_CLAMP5.LS_Adv3 := FALSE;
   S705_LM_DC_2ND_CLAMP5.LS_Ret3 := FALSE;
   S705_LM_DC_2ND_CLAMP5.LS_Adv4 := FALSE;
   S705_LM_DC_2ND_CLAMP5.LS_Ret4 := FALSE;
   S705_LM_DC_2ND_CLAMP5.SOL_Adv := FALSE;
   S705_LM_DC_2ND_CLAMP5.SOL_Ret := FALSE;
   S705_LM_DC_2ND_CLAMP5.M_Ready := TRUE;
   S705_LM_DC_2ND_CLAMP5.T_CHK1 := T#4S;
   S705_LM_DC_2ND_CLAMP5.T_CHK2 := T#4S;
   S705_LM_DC_2ND_CLAMP5.PB_Lamp_CHK := FALSE;
   S705_LM_DC_2ND_CLAMP5.PB_Error_Rst := FALSE;
   S705_LM_DC_2ND_CLAMP5.M_FLICK := TRUE;
   S705_LM_DC_2ND_CLAMP5.M_Adv_Err := FALSE;
   S705_LM_DC_2ND_CLAMP5.M_Ret_Err := FALSE;
   S705_LM_DC_2ND_CLAMP5.LP_Adv := FALSE;
   S705_LM_DC_2ND_CLAMP5.LP_Ret := FALSE;
   S705_LM_DC_2ND_CLAMP5.Visu_Adv := W#16#0;
   S705_LM_DC_2ND_CLAMP5.Visu_Ret := W#16#0;
   S705_LM_DC_2ND_CLAMP5.Error_T1.IN := FALSE;
   S705_LM_DC_2ND_CLAMP5.Error_T1.PT := T#4S;
   S705_LM_DC_2ND_CLAMP5.Error_T1.Q := FALSE;
   S705_LM_DC_2ND_CLAMP5.Error_T1.ET := T#0MS;
   S705_LM_DC_2ND_CLAMP5.Error_T1.STATE := B#16#0;
   S705_LM_DC_2ND_CLAMP5.Error_T1.STIME := T#22D22H55M13S47MS;
   S705_LM_DC_2ND_CLAMP5.Error_T1.ATIME := T#22D22H55M14S365MS;
   S705_LM_DC_2ND_CLAMP5.Error_T2.IN := FALSE;
   S705_LM_DC_2ND_CLAMP5.Error_T2.PT := T#4S;
   S705_LM_DC_2ND_CLAMP5.Error_T2.Q := FALSE;
   S705_LM_DC_2ND_CLAMP5.Error_T2.ET := T#0MS;
   S705_LM_DC_2ND_CLAMP5.Error_T2.STATE := B#16#0;
   S705_LM_DC_2ND_CLAMP5.Error_T2.STIME := T#0MS;
   S705_LM_DC_2ND_CLAMP5.Error_T2.ATIME := T#0MS;
   S705_LM_DC_2ND_CLAMP5.CHK_Aux1 := FALSE;
   S705_LM_DC_2ND_CLAMP5.CHK_Aux2 := FALSE;
   S705_LM_DC_2ND_CLAMP5.Error_T1_DN := FALSE;
   S705_LM_DC_2ND_CLAMP5.Error_T2_DN := FALSE;
   S705_LM_DC_2ND_CLAMP5.Adv_Memo := TRUE;
   S705_LM_DC_2ND_CLAMP5.Visu_Adv_Arr[0] := FALSE;
   S705_LM_DC_2ND_CLAMP5.Visu_Adv_Arr[1] := FALSE;
   S705_LM_DC_2ND_CLAMP5.Visu_Adv_Arr[2] := FALSE;
   S705_LM_DC_2ND_CLAMP5.Visu_Adv_Arr[3] := FALSE;
   S705_LM_DC_2ND_CLAMP5.Visu_Adv_Arr[4] := FALSE;
   S705_LM_DC_2ND_CLAMP5.Visu_Adv_Arr[5] := FALSE;
   S705_LM_DC_2ND_CLAMP5.Visu_Adv_Arr[6] := FALSE;
   S705_LM_DC_2ND_CLAMP5.Visu_Adv_Arr[7] := FALSE;
   S705_LM_DC_2ND_CLAMP5.Visu_Adv_Arr[8] := FALSE;
   S705_LM_DC_2ND_CLAMP5.Visu_Adv_Arr[9] := FALSE;
   S705_LM_DC_2ND_CLAMP5.Visu_Adv_Arr[10] := FALSE;
   S705_LM_DC_2ND_CLAMP5.Visu_Adv_Arr[11] := FALSE;
   S705_LM_DC_2ND_CLAMP5.Visu_Adv_Arr[12] := FALSE;
   S705_LM_DC_2ND_CLAMP5.Visu_Adv_Arr[13] := FALSE;
   S705_LM_DC_2ND_CLAMP5.Visu_Adv_Arr[14] := FALSE;
   S705_LM_DC_2ND_CLAMP5.Visu_Adv_Arr[15] := FALSE;
   S705_LM_DC_2ND_CLAMP5.Visu_Ret_Arr[0] := FALSE;
   S705_LM_DC_2ND_CLAMP5.Visu_Ret_Arr[1] := FALSE;
   S705_LM_DC_2ND_CLAMP5.Visu_Ret_Arr[2] := FALSE;
   S705_LM_DC_2ND_CLAMP5.Visu_Ret_Arr[3] := FALSE;
   S705_LM_DC_2ND_CLAMP5.Visu_Ret_Arr[4] := FALSE;
   S705_LM_DC_2ND_CLAMP5.Visu_Ret_Arr[5] := FALSE;
   S705_LM_DC_2ND_CLAMP5.Visu_Ret_Arr[6] := FALSE;
   S705_LM_DC_2ND_CLAMP5.Visu_Ret_Arr[7] := FALSE;
   S705_LM_DC_2ND_CLAMP5.Visu_Ret_Arr[8] := FALSE;
   S705_LM_DC_2ND_CLAMP5.Visu_Ret_Arr[9] := FALSE;
   S705_LM_DC_2ND_CLAMP5.Visu_Ret_Arr[10] := FALSE;
   S705_LM_DC_2ND_CLAMP5.Visu_Ret_Arr[11] := FALSE;
   S705_LM_DC_2ND_CLAMP5.Visu_Ret_Arr[12] := FALSE;
   S705_LM_DC_2ND_CLAMP5.Visu_Ret_Arr[13] := FALSE;
   S705_LM_DC_2ND_CLAMP5.Visu_Ret_Arr[14] := FALSE;
   S705_LM_DC_2ND_CLAMP5.Visu_Ret_Arr[15] := FALSE;
   S705_LM_DC_2ND_CLAMP5.BLK_Move_Ret := 0;
   S705_LM_DC_2ND_CLAMP5.Enable := FALSE;
   S705_LM_DC_2ND_CLAMP5.Adv_End := FALSE;
   S705_LM_DC_2ND_CLAMP5.Ret_End := FALSE;
   S705_LM_DC_STK_PIN.Enable_Aux := FALSE;
   S705_LM_DC_STK_PIN.Adv_Amount := 1;
   S705_LM_DC_STK_PIN.Ret_Amount := 1;
   S705_LM_DC_STK_PIN.LS_Adv1 := FALSE;
   S705_LM_DC_STK_PIN.LS_Ret1 := FALSE;
   S705_LM_DC_STK_PIN.LS_Adv2 := FALSE;
   S705_LM_DC_STK_PIN.LS_Ret2 := FALSE;
   S705_LM_DC_STK_PIN.LS_Adv3 := FALSE;
   S705_LM_DC_STK_PIN.LS_Ret3 := FALSE;
   S705_LM_DC_STK_PIN.LS_Adv4 := FALSE;
   S705_LM_DC_STK_PIN.LS_Ret4 := FALSE;
   S705_LM_DC_STK_PIN.SOL_Adv := FALSE;
   S705_LM_DC_STK_PIN.SOL_Ret := FALSE;
   S705_LM_DC_STK_PIN.M_Ready := TRUE;
   S705_LM_DC_STK_PIN.T_CHK1 := T#4S;
   S705_LM_DC_STK_PIN.T_CHK2 := T#4S;
   S705_LM_DC_STK_PIN.PB_Lamp_CHK := FALSE;
   S705_LM_DC_STK_PIN.PB_Error_Rst := FALSE;
   S705_LM_DC_STK_PIN.M_FLICK := TRUE;
   S705_LM_DC_STK_PIN.M_Adv_Err := FALSE;
   S705_LM_DC_STK_PIN.M_Ret_Err := FALSE;
   S705_LM_DC_STK_PIN.LP_Adv := FALSE;
   S705_LM_DC_STK_PIN.LP_Ret := FALSE;
   S705_LM_DC_STK_PIN.Visu_Adv := W#16#0;
   S705_LM_DC_STK_PIN.Visu_Ret := W#16#0;
   S705_LM_DC_STK_PIN.Error_T1.IN := FALSE;
   S705_LM_DC_STK_PIN.Error_T1.PT := T#4S;
   S705_LM_DC_STK_PIN.Error_T1.Q := FALSE;
   S705_LM_DC_STK_PIN.Error_T1.ET := T#0MS;
   S705_LM_DC_STK_PIN.Error_T1.STATE := B#16#0;
   S705_LM_DC_STK_PIN.Error_T1.STIME := T#14D12H57M37S831MS;
   S705_LM_DC_STK_PIN.Error_T1.ATIME := T#14D12H57M37S878MS;
   S705_LM_DC_STK_PIN.Error_T2.IN := FALSE;
   S705_LM_DC_STK_PIN.Error_T2.PT := T#4S;
   S705_LM_DC_STK_PIN.Error_T2.Q := FALSE;
   S705_LM_DC_STK_PIN.Error_T2.ET := T#0MS;
   S705_LM_DC_STK_PIN.Error_T2.STATE := B#16#0;
   S705_LM_DC_STK_PIN.Error_T2.STIME := T#0MS;
   S705_LM_DC_STK_PIN.Error_T2.ATIME := T#0MS;
   S705_LM_DC_STK_PIN.CHK_Aux1 := FALSE;
   S705_LM_DC_STK_PIN.CHK_Aux2 := FALSE;
   S705_LM_DC_STK_PIN.Error_T1_DN := FALSE;
   S705_LM_DC_STK_PIN.Error_T2_DN := FALSE;
   S705_LM_DC_STK_PIN.Adv_Memo := FALSE;
   S705_LM_DC_STK_PIN.Visu_Adv_Arr[0] := FALSE;
   S705_LM_DC_STK_PIN.Visu_Adv_Arr[1] := FALSE;
   S705_LM_DC_STK_PIN.Visu_Adv_Arr[2] := FALSE;
   S705_LM_DC_STK_PIN.Visu_Adv_Arr[3] := FALSE;
   S705_LM_DC_STK_PIN.Visu_Adv_Arr[4] := FALSE;
   S705_LM_DC_STK_PIN.Visu_Adv_Arr[5] := FALSE;
   S705_LM_DC_STK_PIN.Visu_Adv_Arr[6] := FALSE;
   S705_LM_DC_STK_PIN.Visu_Adv_Arr[7] := FALSE;
   S705_LM_DC_STK_PIN.Visu_Adv_Arr[8] := FALSE;
   S705_LM_DC_STK_PIN.Visu_Adv_Arr[9] := FALSE;
   S705_LM_DC_STK_PIN.Visu_Adv_Arr[10] := FALSE;
   S705_LM_DC_STK_PIN.Visu_Adv_Arr[11] := FALSE;
   S705_LM_DC_STK_PIN.Visu_Adv_Arr[12] := FALSE;
   S705_LM_DC_STK_PIN.Visu_Adv_Arr[13] := FALSE;
   S705_LM_DC_STK_PIN.Visu_Adv_Arr[14] := FALSE;
   S705_LM_DC_STK_PIN.Visu_Adv_Arr[15] := FALSE;
   S705_LM_DC_STK_PIN.Visu_Ret_Arr[0] := FALSE;
   S705_LM_DC_STK_PIN.Visu_Ret_Arr[1] := FALSE;
   S705_LM_DC_STK_PIN.Visu_Ret_Arr[2] := FALSE;
   S705_LM_DC_STK_PIN.Visu_Ret_Arr[3] := FALSE;
   S705_LM_DC_STK_PIN.Visu_Ret_Arr[4] := FALSE;
   S705_LM_DC_STK_PIN.Visu_Ret_Arr[5] := FALSE;
   S705_LM_DC_STK_PIN.Visu_Ret_Arr[6] := FALSE;
   S705_LM_DC_STK_PIN.Visu_Ret_Arr[7] := FALSE;
   S705_LM_DC_STK_PIN.Visu_Ret_Arr[8] := FALSE;
   S705_LM_DC_STK_PIN.Visu_Ret_Arr[9] := FALSE;
   S705_LM_DC_STK_PIN.Visu_Ret_Arr[10] := FALSE;
   S705_LM_DC_STK_PIN.Visu_Ret_Arr[11] := FALSE;
   S705_LM_DC_STK_PIN.Visu_Ret_Arr[12] := FALSE;
   S705_LM_DC_STK_PIN.Visu_Ret_Arr[13] := FALSE;
   S705_LM_DC_STK_PIN.Visu_Ret_Arr[14] := FALSE;
   S705_LM_DC_STK_PIN.Visu_Ret_Arr[15] := FALSE;
   S705_LM_DC_STK_PIN.BLK_Move_Ret := 0;
   S705_LM_DC_STK_PIN.Enable := FALSE;
   S705_LM_DC_STK_PIN.Adv_End := FALSE;
   S705_LM_DC_STK_PIN.Ret_End := FALSE;
   S705_LM_DC_OTR_CLAMP.Enable_Aux := FALSE;
   S705_LM_DC_OTR_CLAMP.Adv_Amount := 1;
   S705_LM_DC_OTR_CLAMP.Ret_Amount := 1;
   S705_LM_DC_OTR_CLAMP.LS_Adv1 := FALSE;
   S705_LM_DC_OTR_CLAMP.LS_Ret1 := FALSE;
   S705_LM_DC_OTR_CLAMP.LS_Adv2 := FALSE;
   S705_LM_DC_OTR_CLAMP.LS_Ret2 := FALSE;
   S705_LM_DC_OTR_CLAMP.LS_Adv3 := FALSE;
   S705_LM_DC_OTR_CLAMP.LS_Ret3 := FALSE;
   S705_LM_DC_OTR_CLAMP.LS_Adv4 := FALSE;
   S705_LM_DC_OTR_CLAMP.LS_Ret4 := FALSE;
   S705_LM_DC_OTR_CLAMP.SOL_Adv := FALSE;
   S705_LM_DC_OTR_CLAMP.SOL_Ret := FALSE;
   S705_LM_DC_OTR_CLAMP.M_Ready := TRUE;
   S705_LM_DC_OTR_CLAMP.T_CHK1 := T#4S;
   S705_LM_DC_OTR_CLAMP.T_CHK2 := T#4S;
   S705_LM_DC_OTR_CLAMP.PB_Lamp_CHK := FALSE;
   S705_LM_DC_OTR_CLAMP.PB_Error_Rst := FALSE;
   S705_LM_DC_OTR_CLAMP.M_FLICK := TRUE;
   S705_LM_DC_OTR_CLAMP.M_Adv_Err := FALSE;
   S705_LM_DC_OTR_CLAMP.M_Ret_Err := FALSE;
   S705_LM_DC_OTR_CLAMP.LP_Adv := FALSE;
   S705_LM_DC_OTR_CLAMP.LP_Ret := FALSE;
   S705_LM_DC_OTR_CLAMP.Visu_Adv := W#16#0;
   S705_LM_DC_OTR_CLAMP.Visu_Ret := W#16#0;
   S705_LM_DC_OTR_CLAMP.Error_T1.IN := FALSE;
   S705_LM_DC_OTR_CLAMP.Error_T1.PT := T#4S;
   S705_LM_DC_OTR_CLAMP.Error_T1.Q := FALSE;
   S705_LM_DC_OTR_CLAMP.Error_T1.ET := T#0MS;
   S705_LM_DC_OTR_CLAMP.Error_T1.STATE := B#16#0;
   S705_LM_DC_OTR_CLAMP.Error_T1.STIME := T#14D12H57M37S831MS;
   S705_LM_DC_OTR_CLAMP.Error_T1.ATIME := T#14D12H57M37S878MS;
   S705_LM_DC_OTR_CLAMP.Error_T2.IN := FALSE;
   S705_LM_DC_OTR_CLAMP.Error_T2.PT := T#4S;
   S705_LM_DC_OTR_CLAMP.Error_T2.Q := FALSE;
   S705_LM_DC_OTR_CLAMP.Error_T2.ET := T#0MS;
   S705_LM_DC_OTR_CLAMP.Error_T2.STATE := B#16#0;
   S705_LM_DC_OTR_CLAMP.Error_T2.STIME := T#0MS;
   S705_LM_DC_OTR_CLAMP.Error_T2.ATIME := T#0MS;
   S705_LM_DC_OTR_CLAMP.CHK_Aux1 := FALSE;
   S705_LM_DC_OTR_CLAMP.CHK_Aux2 := FALSE;
   S705_LM_DC_OTR_CLAMP.Error_T1_DN := FALSE;
   S705_LM_DC_OTR_CLAMP.Error_T2_DN := FALSE;
   S705_LM_DC_OTR_CLAMP.Adv_Memo := FALSE;
   S705_LM_DC_OTR_CLAMP.Visu_Adv_Arr[0] := FALSE;
   S705_LM_DC_OTR_CLAMP.Visu_Adv_Arr[1] := FALSE;
   S705_LM_DC_OTR_CLAMP.Visu_Adv_Arr[2] := FALSE;
   S705_LM_DC_OTR_CLAMP.Visu_Adv_Arr[3] := FALSE;
   S705_LM_DC_OTR_CLAMP.Visu_Adv_Arr[4] := FALSE;
   S705_LM_DC_OTR_CLAMP.Visu_Adv_Arr[5] := FALSE;
   S705_LM_DC_OTR_CLAMP.Visu_Adv_Arr[6] := FALSE;
   S705_LM_DC_OTR_CLAMP.Visu_Adv_Arr[7] := FALSE;
   S705_LM_DC_OTR_CLAMP.Visu_Adv_Arr[8] := FALSE;
   S705_LM_DC_OTR_CLAMP.Visu_Adv_Arr[9] := FALSE;
   S705_LM_DC_OTR_CLAMP.Visu_Adv_Arr[10] := FALSE;
   S705_LM_DC_OTR_CLAMP.Visu_Adv_Arr[11] := FALSE;
   S705_LM_DC_OTR_CLAMP.Visu_Adv_Arr[12] := FALSE;
   S705_LM_DC_OTR_CLAMP.Visu_Adv_Arr[13] := FALSE;
   S705_LM_DC_OTR_CLAMP.Visu_Adv_Arr[14] := FALSE;
   S705_LM_DC_OTR_CLAMP.Visu_Adv_Arr[15] := FALSE;
   S705_LM_DC_OTR_CLAMP.Visu_Ret_Arr[0] := FALSE;
   S705_LM_DC_OTR_CLAMP.Visu_Ret_Arr[1] := FALSE;
   S705_LM_DC_OTR_CLAMP.Visu_Ret_Arr[2] := FALSE;
   S705_LM_DC_OTR_CLAMP.Visu_Ret_Arr[3] := FALSE;
   S705_LM_DC_OTR_CLAMP.Visu_Ret_Arr[4] := FALSE;
   S705_LM_DC_OTR_CLAMP.Visu_Ret_Arr[5] := FALSE;
   S705_LM_DC_OTR_CLAMP.Visu_Ret_Arr[6] := FALSE;
   S705_LM_DC_OTR_CLAMP.Visu_Ret_Arr[7] := FALSE;
   S705_LM_DC_OTR_CLAMP.Visu_Ret_Arr[8] := FALSE;
   S705_LM_DC_OTR_CLAMP.Visu_Ret_Arr[9] := FALSE;
   S705_LM_DC_OTR_CLAMP.Visu_Ret_Arr[10] := FALSE;
   S705_LM_DC_OTR_CLAMP.Visu_Ret_Arr[11] := FALSE;
   S705_LM_DC_OTR_CLAMP.Visu_Ret_Arr[12] := FALSE;
   S705_LM_DC_OTR_CLAMP.Visu_Ret_Arr[13] := FALSE;
   S705_LM_DC_OTR_CLAMP.Visu_Ret_Arr[14] := FALSE;
   S705_LM_DC_OTR_CLAMP.Visu_Ret_Arr[15] := FALSE;
   S705_LM_DC_OTR_CLAMP.BLK_Move_Ret := 0;
   S705_LM_DC_OTR_CLAMP.Enable := FALSE;
   S705_LM_DC_OTR_CLAMP.Adv_End := FALSE;
   S705_LM_DC_OTR_CLAMP.Ret_End := FALSE;
   S705_LM_DC_ASSY_CLAMP.Enable_Aux := FALSE;
   S705_LM_DC_ASSY_CLAMP.Adv_Amount := 1;
   S705_LM_DC_ASSY_CLAMP.Ret_Amount := 1;
   S705_LM_DC_ASSY_CLAMP.LS_Adv1 := FALSE;
   S705_LM_DC_ASSY_CLAMP.LS_Ret1 := FALSE;
   S705_LM_DC_ASSY_CLAMP.LS_Adv2 := FALSE;
   S705_LM_DC_ASSY_CLAMP.LS_Ret2 := FALSE;
   S705_LM_DC_ASSY_CLAMP.LS_Adv3 := FALSE;
   S705_LM_DC_ASSY_CLAMP.LS_Ret3 := FALSE;
   S705_LM_DC_ASSY_CLAMP.LS_Adv4 := FALSE;
   S705_LM_DC_ASSY_CLAMP.LS_Ret4 := FALSE;
   S705_LM_DC_ASSY_CLAMP.SOL_Adv := FALSE;
   S705_LM_DC_ASSY_CLAMP.SOL_Ret := FALSE;
   S705_LM_DC_ASSY_CLAMP.M_Ready := TRUE;
   S705_LM_DC_ASSY_CLAMP.T_CHK1 := T#4S;
   S705_LM_DC_ASSY_CLAMP.T_CHK2 := T#4S;
   S705_LM_DC_ASSY_CLAMP.PB_Lamp_CHK := FALSE;
   S705_LM_DC_ASSY_CLAMP.PB_Error_Rst := FALSE;
   S705_LM_DC_ASSY_CLAMP.M_FLICK := TRUE;
   S705_LM_DC_ASSY_CLAMP.M_Adv_Err := FALSE;
   S705_LM_DC_ASSY_CLAMP.M_Ret_Err := FALSE;
   S705_LM_DC_ASSY_CLAMP.LP_Adv := FALSE;
   S705_LM_DC_ASSY_CLAMP.LP_Ret := FALSE;
   S705_LM_DC_ASSY_CLAMP.Visu_Adv := W#16#0;
   S705_LM_DC_ASSY_CLAMP.Visu_Ret := W#16#0;
   S705_LM_DC_ASSY_CLAMP.Error_T1.IN := FALSE;
   S705_LM_DC_ASSY_CLAMP.Error_T1.PT := T#4S;
   S705_LM_DC_ASSY_CLAMP.Error_T1.Q := FALSE;
   S705_LM_DC_ASSY_CLAMP.Error_T1.ET := T#0MS;
   S705_LM_DC_ASSY_CLAMP.Error_T1.STATE := B#16#0;
   S705_LM_DC_ASSY_CLAMP.Error_T1.STIME := T#22D22H55M12S68MS;
   S705_LM_DC_ASSY_CLAMP.Error_T1.ATIME := T#22D22H55M13S;
   S705_LM_DC_ASSY_CLAMP.Error_T2.IN := FALSE;
   S705_LM_DC_ASSY_CLAMP.Error_T2.PT := T#4S;
   S705_LM_DC_ASSY_CLAMP.Error_T2.Q := FALSE;
   S705_LM_DC_ASSY_CLAMP.Error_T2.ET := T#0MS;
   S705_LM_DC_ASSY_CLAMP.Error_T2.STATE := B#16#0;
   S705_LM_DC_ASSY_CLAMP.Error_T2.STIME := T#0MS;
   S705_LM_DC_ASSY_CLAMP.Error_T2.ATIME := T#0MS;
   S705_LM_DC_ASSY_CLAMP.CHK_Aux1 := FALSE;
   S705_LM_DC_ASSY_CLAMP.CHK_Aux2 := FALSE;
   S705_LM_DC_ASSY_CLAMP.Error_T1_DN := FALSE;
   S705_LM_DC_ASSY_CLAMP.Error_T2_DN := FALSE;
   S705_LM_DC_ASSY_CLAMP.Adv_Memo := TRUE;
   S705_LM_DC_ASSY_CLAMP.Visu_Adv_Arr[0] := FALSE;
   S705_LM_DC_ASSY_CLAMP.Visu_Adv_Arr[1] := FALSE;
   S705_LM_DC_ASSY_CLAMP.Visu_Adv_Arr[2] := FALSE;
   S705_LM_DC_ASSY_CLAMP.Visu_Adv_Arr[3] := FALSE;
   S705_LM_DC_ASSY_CLAMP.Visu_Adv_Arr[4] := FALSE;
   S705_LM_DC_ASSY_CLAMP.Visu_Adv_Arr[5] := FALSE;
   S705_LM_DC_ASSY_CLAMP.Visu_Adv_Arr[6] := FALSE;
   S705_LM_DC_ASSY_CLAMP.Visu_Adv_Arr[7] := FALSE;
   S705_LM_DC_ASSY_CLAMP.Visu_Adv_Arr[8] := FALSE;
   S705_LM_DC_ASSY_CLAMP.Visu_Adv_Arr[9] := FALSE;
   S705_LM_DC_ASSY_CLAMP.Visu_Adv_Arr[10] := FALSE;
   S705_LM_DC_ASSY_CLAMP.Visu_Adv_Arr[11] := FALSE;
   S705_LM_DC_ASSY_CLAMP.Visu_Adv_Arr[12] := FALSE;
   S705_LM_DC_ASSY_CLAMP.Visu_Adv_Arr[13] := FALSE;
   S705_LM_DC_ASSY_CLAMP.Visu_Adv_Arr[14] := FALSE;
   S705_LM_DC_ASSY_CLAMP.Visu_Adv_Arr[15] := FALSE;
   S705_LM_DC_ASSY_CLAMP.Visu_Ret_Arr[0] := FALSE;
   S705_LM_DC_ASSY_CLAMP.Visu_Ret_Arr[1] := FALSE;
   S705_LM_DC_ASSY_CLAMP.Visu_Ret_Arr[2] := FALSE;
   S705_LM_DC_ASSY_CLAMP.Visu_Ret_Arr[3] := FALSE;
   S705_LM_DC_ASSY_CLAMP.Visu_Ret_Arr[4] := FALSE;
   S705_LM_DC_ASSY_CLAMP.Visu_Ret_Arr[5] := FALSE;
   S705_LM_DC_ASSY_CLAMP.Visu_Ret_Arr[6] := FALSE;
   S705_LM_DC_ASSY_CLAMP.Visu_Ret_Arr[7] := FALSE;
   S705_LM_DC_ASSY_CLAMP.Visu_Ret_Arr[8] := FALSE;
   S705_LM_DC_ASSY_CLAMP.Visu_Ret_Arr[9] := FALSE;
   S705_LM_DC_ASSY_CLAMP.Visu_Ret_Arr[10] := FALSE;
   S705_LM_DC_ASSY_CLAMP.Visu_Ret_Arr[11] := FALSE;
   S705_LM_DC_ASSY_CLAMP.Visu_Ret_Arr[12] := FALSE;
   S705_LM_DC_ASSY_CLAMP.Visu_Ret_Arr[13] := FALSE;
   S705_LM_DC_ASSY_CLAMP.Visu_Ret_Arr[14] := FALSE;
   S705_LM_DC_ASSY_CLAMP.Visu_Ret_Arr[15] := FALSE;
   S705_LM_DC_ASSY_CLAMP.BLK_Move_Ret := 0;
   S705_LM_DC_ASSY_CLAMP.Enable := FALSE;
   S705_LM_DC_ASSY_CLAMP.Adv_End := FALSE;
   S705_LM_DC_ASSY_CLAMP.Ret_End := FALSE;
   S705_LM_DC_FF_PIN.Enable_Aux := FALSE;
   S705_LM_DC_FF_PIN.Adv_Amount := 1;
   S705_LM_DC_FF_PIN.Ret_Amount := 1;
   S705_LM_DC_FF_PIN.LS_Adv1 := FALSE;
   S705_LM_DC_FF_PIN.LS_Ret1 := FALSE;
   S705_LM_DC_FF_PIN.LS_Adv2 := FALSE;
   S705_LM_DC_FF_PIN.LS_Ret2 := FALSE;
   S705_LM_DC_FF_PIN.LS_Adv3 := FALSE;
   S705_LM_DC_FF_PIN.LS_Ret3 := FALSE;
   S705_LM_DC_FF_PIN.LS_Adv4 := FALSE;
   S705_LM_DC_FF_PIN.LS_Ret4 := FALSE;
   S705_LM_DC_FF_PIN.SOL_Adv := FALSE;
   S705_LM_DC_FF_PIN.SOL_Ret := FALSE;
   S705_LM_DC_FF_PIN.M_Ready := TRUE;
   S705_LM_DC_FF_PIN.T_CHK1 := T#4S;
   S705_LM_DC_FF_PIN.T_CHK2 := T#4S;
   S705_LM_DC_FF_PIN.PB_Lamp_CHK := FALSE;
   S705_LM_DC_FF_PIN.PB_Error_Rst := FALSE;
   S705_LM_DC_FF_PIN.M_FLICK := TRUE;
   S705_LM_DC_FF_PIN.M_Adv_Err := FALSE;
   S705_LM_DC_FF_PIN.M_Ret_Err := FALSE;
   S705_LM_DC_FF_PIN.LP_Adv := FALSE;
   S705_LM_DC_FF_PIN.LP_Ret := FALSE;
   S705_LM_DC_FF_PIN.Visu_Adv := W#16#0;
   S705_LM_DC_FF_PIN.Visu_Ret := W#16#0;
   S705_LM_DC_FF_PIN.Error_T1.IN := FALSE;
   S705_LM_DC_FF_PIN.Error_T1.PT := T#4S;
   S705_LM_DC_FF_PIN.Error_T1.Q := FALSE;
   S705_LM_DC_FF_PIN.Error_T1.ET := T#0MS;
   S705_LM_DC_FF_PIN.Error_T1.STATE := B#16#0;
   S705_LM_DC_FF_PIN.Error_T1.STIME := T#14D12H57M37S831MS;
   S705_LM_DC_FF_PIN.Error_T1.ATIME := T#14D12H57M37S878MS;
   S705_LM_DC_FF_PIN.Error_T2.IN := FALSE;
   S705_LM_DC_FF_PIN.Error_T2.PT := T#4S;
   S705_LM_DC_FF_PIN.Error_T2.Q := FALSE;
   S705_LM_DC_FF_PIN.Error_T2.ET := T#0MS;
   S705_LM_DC_FF_PIN.Error_T2.STATE := B#16#0;
   S705_LM_DC_FF_PIN.Error_T2.STIME := T#0MS;
   S705_LM_DC_FF_PIN.Error_T2.ATIME := T#0MS;
   S705_LM_DC_FF_PIN.CHK_Aux1 := FALSE;
   S705_LM_DC_FF_PIN.CHK_Aux2 := FALSE;
   S705_LM_DC_FF_PIN.Error_T1_DN := FALSE;
   S705_LM_DC_FF_PIN.Error_T2_DN := FALSE;
   S705_LM_DC_FF_PIN.Adv_Memo := FALSE;
   S705_LM_DC_FF_PIN.Visu_Adv_Arr[0] := FALSE;
   S705_LM_DC_FF_PIN.Visu_Adv_Arr[1] := FALSE;
   S705_LM_DC_FF_PIN.Visu_Adv_Arr[2] := FALSE;
   S705_LM_DC_FF_PIN.Visu_Adv_Arr[3] := FALSE;
   S705_LM_DC_FF_PIN.Visu_Adv_Arr[4] := FALSE;
   S705_LM_DC_FF_PIN.Visu_Adv_Arr[5] := FALSE;
   S705_LM_DC_FF_PIN.Visu_Adv_Arr[6] := FALSE;
   S705_LM_DC_FF_PIN.Visu_Adv_Arr[7] := FALSE;
   S705_LM_DC_FF_PIN.Visu_Adv_Arr[8] := FALSE;
   S705_LM_DC_FF_PIN.Visu_Adv_Arr[9] := FALSE;
   S705_LM_DC_FF_PIN.Visu_Adv_Arr[10] := FALSE;
   S705_LM_DC_FF_PIN.Visu_Adv_Arr[11] := FALSE;
   S705_LM_DC_FF_PIN.Visu_Adv_Arr[12] := FALSE;
   S705_LM_DC_FF_PIN.Visu_Adv_Arr[13] := FALSE;
   S705_LM_DC_FF_PIN.Visu_Adv_Arr[14] := FALSE;
   S705_LM_DC_FF_PIN.Visu_Adv_Arr[15] := FALSE;
   S705_LM_DC_FF_PIN.Visu_Ret_Arr[0] := FALSE;
   S705_LM_DC_FF_PIN.Visu_Ret_Arr[1] := FALSE;
   S705_LM_DC_FF_PIN.Visu_Ret_Arr[2] := FALSE;
   S705_LM_DC_FF_PIN.Visu_Ret_Arr[3] := FALSE;
   S705_LM_DC_FF_PIN.Visu_Ret_Arr[4] := FALSE;
   S705_LM_DC_FF_PIN.Visu_Ret_Arr[5] := FALSE;
   S705_LM_DC_FF_PIN.Visu_Ret_Arr[6] := FALSE;
   S705_LM_DC_FF_PIN.Visu_Ret_Arr[7] := FALSE;
   S705_LM_DC_FF_PIN.Visu_Ret_Arr[8] := FALSE;
   S705_LM_DC_FF_PIN.Visu_Ret_Arr[9] := FALSE;
   S705_LM_DC_FF_PIN.Visu_Ret_Arr[10] := FALSE;
   S705_LM_DC_FF_PIN.Visu_Ret_Arr[11] := FALSE;
   S705_LM_DC_FF_PIN.Visu_Ret_Arr[12] := FALSE;
   S705_LM_DC_FF_PIN.Visu_Ret_Arr[13] := FALSE;
   S705_LM_DC_FF_PIN.Visu_Ret_Arr[14] := FALSE;
   S705_LM_DC_FF_PIN.Visu_Ret_Arr[15] := FALSE;
   S705_LM_DC_FF_PIN.BLK_Move_Ret := 0;
   S705_LM_DC_FF_PIN.Enable := FALSE;
   S705_LM_DC_FF_PIN.Adv_End := FALSE;
   S705_LM_DC_FF_PIN.Ret_End := FALSE;
   S705_LM_DC_FF_CLAMP.Enable_Aux := FALSE;
   S705_LM_DC_FF_CLAMP.Adv_Amount := 1;
   S705_LM_DC_FF_CLAMP.Ret_Amount := 1;
   S705_LM_DC_FF_CLAMP.LS_Adv1 := FALSE;
   S705_LM_DC_FF_CLAMP.LS_Ret1 := FALSE;
   S705_LM_DC_FF_CLAMP.LS_Adv2 := FALSE;
   S705_LM_DC_FF_CLAMP.LS_Ret2 := FALSE;
   S705_LM_DC_FF_CLAMP.LS_Adv3 := FALSE;
   S705_LM_DC_FF_CLAMP.LS_Ret3 := FALSE;
   S705_LM_DC_FF_CLAMP.LS_Adv4 := FALSE;
   S705_LM_DC_FF_CLAMP.LS_Ret4 := FALSE;
   S705_LM_DC_FF_CLAMP.SOL_Adv := FALSE;
   S705_LM_DC_FF_CLAMP.SOL_Ret := FALSE;
   S705_LM_DC_FF_CLAMP.M_Ready := TRUE;
   S705_LM_DC_FF_CLAMP.T_CHK1 := T#4S;
   S705_LM_DC_FF_CLAMP.T_CHK2 := T#4S;
   S705_LM_DC_FF_CLAMP.PB_Lamp_CHK := FALSE;
   S705_LM_DC_FF_CLAMP.PB_Error_Rst := FALSE;
   S705_LM_DC_FF_CLAMP.M_FLICK := TRUE;
   S705_LM_DC_FF_CLAMP.M_Adv_Err := FALSE;
   S705_LM_DC_FF_CLAMP.M_Ret_Err := FALSE;
   S705_LM_DC_FF_CLAMP.LP_Adv := FALSE;
   S705_LM_DC_FF_CLAMP.LP_Ret := FALSE;
   S705_LM_DC_FF_CLAMP.Visu_Adv := W#16#0;
   S705_LM_DC_FF_CLAMP.Visu_Ret := W#16#0;
   S705_LM_DC_FF_CLAMP.Error_T1.IN := FALSE;
   S705_LM_DC_FF_CLAMP.Error_T1.PT := T#4S;
   S705_LM_DC_FF_CLAMP.Error_T1.Q := FALSE;
   S705_LM_DC_FF_CLAMP.Error_T1.ET := T#0MS;
   S705_LM_DC_FF_CLAMP.Error_T1.STATE := B#16#0;
   S705_LM_DC_FF_CLAMP.Error_T1.STIME := T#14D12H57M37S831MS;
   S705_LM_DC_FF_CLAMP.Error_T1.ATIME := T#14D12H57M37S878MS;
   S705_LM_DC_FF_CLAMP.Error_T2.IN := FALSE;
   S705_LM_DC_FF_CLAMP.Error_T2.PT := T#4S;
   S705_LM_DC_FF_CLAMP.Error_T2.Q := FALSE;
   S705_LM_DC_FF_CLAMP.Error_T2.ET := T#0MS;
   S705_LM_DC_FF_CLAMP.Error_T2.STATE := B#16#0;
   S705_LM_DC_FF_CLAMP.Error_T2.STIME := T#0MS;
   S705_LM_DC_FF_CLAMP.Error_T2.ATIME := T#0MS;
   S705_LM_DC_FF_CLAMP.CHK_Aux1 := FALSE;
   S705_LM_DC_FF_CLAMP.CHK_Aux2 := FALSE;
   S705_LM_DC_FF_CLAMP.Error_T1_DN := FALSE;
   S705_LM_DC_FF_CLAMP.Error_T2_DN := FALSE;
   S705_LM_DC_FF_CLAMP.Adv_Memo := FALSE;
   S705_LM_DC_FF_CLAMP.Visu_Adv_Arr[0] := FALSE;
   S705_LM_DC_FF_CLAMP.Visu_Adv_Arr[1] := FALSE;
   S705_LM_DC_FF_CLAMP.Visu_Adv_Arr[2] := FALSE;
   S705_LM_DC_FF_CLAMP.Visu_Adv_Arr[3] := FALSE;
   S705_LM_DC_FF_CLAMP.Visu_Adv_Arr[4] := FALSE;
   S705_LM_DC_FF_CLAMP.Visu_Adv_Arr[5] := FALSE;
   S705_LM_DC_FF_CLAMP.Visu_Adv_Arr[6] := FALSE;
   S705_LM_DC_FF_CLAMP.Visu_Adv_Arr[7] := FALSE;
   S705_LM_DC_FF_CLAMP.Visu_Adv_Arr[8] := FALSE;
   S705_LM_DC_FF_CLAMP.Visu_Adv_Arr[9] := FALSE;
   S705_LM_DC_FF_CLAMP.Visu_Adv_Arr[10] := FALSE;
   S705_LM_DC_FF_CLAMP.Visu_Adv_Arr[11] := FALSE;
   S705_LM_DC_FF_CLAMP.Visu_Adv_Arr[12] := FALSE;
   S705_LM_DC_FF_CLAMP.Visu_Adv_Arr[13] := FALSE;
   S705_LM_DC_FF_CLAMP.Visu_Adv_Arr[14] := FALSE;
   S705_LM_DC_FF_CLAMP.Visu_Adv_Arr[15] := FALSE;
   S705_LM_DC_FF_CLAMP.Visu_Ret_Arr[0] := FALSE;
   S705_LM_DC_FF_CLAMP.Visu_Ret_Arr[1] := FALSE;
   S705_LM_DC_FF_CLAMP.Visu_Ret_Arr[2] := FALSE;
   S705_LM_DC_FF_CLAMP.Visu_Ret_Arr[3] := FALSE;
   S705_LM_DC_FF_CLAMP.Visu_Ret_Arr[4] := FALSE;
   S705_LM_DC_FF_CLAMP.Visu_Ret_Arr[5] := FALSE;
   S705_LM_DC_FF_CLAMP.Visu_Ret_Arr[6] := FALSE;
   S705_LM_DC_FF_CLAMP.Visu_Ret_Arr[7] := FALSE;
   S705_LM_DC_FF_CLAMP.Visu_Ret_Arr[8] := FALSE;
   S705_LM_DC_FF_CLAMP.Visu_Ret_Arr[9] := FALSE;
   S705_LM_DC_FF_CLAMP.Visu_Ret_Arr[10] := FALSE;
   S705_LM_DC_FF_CLAMP.Visu_Ret_Arr[11] := FALSE;
   S705_LM_DC_FF_CLAMP.Visu_Ret_Arr[12] := FALSE;
   S705_LM_DC_FF_CLAMP.Visu_Ret_Arr[13] := FALSE;
   S705_LM_DC_FF_CLAMP.Visu_Ret_Arr[14] := FALSE;
   S705_LM_DC_FF_CLAMP.Visu_Ret_Arr[15] := FALSE;
   S705_LM_DC_FF_CLAMP.BLK_Move_Ret := 0;
   S705_LM_DC_FF_CLAMP.Enable := FALSE;
   S705_LM_DC_FF_CLAMP.Adv_End := FALSE;
   S705_LM_DC_FF_CLAMP.Ret_End := FALSE;
   S705_LM_DC_2ND_CLAMP6.Enable_Aux := FALSE;
   S705_LM_DC_2ND_CLAMP6.Adv_Amount := 2;
   S705_LM_DC_2ND_CLAMP6.Ret_Amount := 2;
   S705_LM_DC_2ND_CLAMP6.LS_Adv1 := FALSE;
   S705_LM_DC_2ND_CLAMP6.LS_Ret1 := FALSE;
   S705_LM_DC_2ND_CLAMP6.LS_Adv2 := FALSE;
   S705_LM_DC_2ND_CLAMP6.LS_Ret2 := FALSE;
   S705_LM_DC_2ND_CLAMP6.LS_Adv3 := FALSE;
   S705_LM_DC_2ND_CLAMP6.LS_Ret3 := FALSE;
   S705_LM_DC_2ND_CLAMP6.LS_Adv4 := FALSE;
   S705_LM_DC_2ND_CLAMP6.LS_Ret4 := FALSE;
   S705_LM_DC_2ND_CLAMP6.SOL_Adv := FALSE;
   S705_LM_DC_2ND_CLAMP6.SOL_Ret := FALSE;
   S705_LM_DC_2ND_CLAMP6.M_Ready := TRUE;
   S705_LM_DC_2ND_CLAMP6.T_CHK1 := T#4S;
   S705_LM_DC_2ND_CLAMP6.T_CHK2 := T#4S;
   S705_LM_DC_2ND_CLAMP6.PB_Lamp_CHK := FALSE;
   S705_LM_DC_2ND_CLAMP6.PB_Error_Rst := FALSE;
   S705_LM_DC_2ND_CLAMP6.M_FLICK := TRUE;
   S705_LM_DC_2ND_CLAMP6.M_Adv_Err := FALSE;
   S705_LM_DC_2ND_CLAMP6.M_Ret_Err := FALSE;
   S705_LM_DC_2ND_CLAMP6.LP_Adv := FALSE;
   S705_LM_DC_2ND_CLAMP6.LP_Ret := FALSE;
   S705_LM_DC_2ND_CLAMP6.Visu_Adv := W#16#0;
   S705_LM_DC_2ND_CLAMP6.Visu_Ret := W#16#0;
   S705_LM_DC_2ND_CLAMP6.Error_T1.IN := FALSE;
   S705_LM_DC_2ND_CLAMP6.Error_T1.PT := T#4S;
   S705_LM_DC_2ND_CLAMP6.Error_T1.Q := FALSE;
   S705_LM_DC_2ND_CLAMP6.Error_T1.ET := T#0MS;
   S705_LM_DC_2ND_CLAMP6.Error_T1.STATE := B#16#0;
   S705_LM_DC_2ND_CLAMP6.Error_T1.STIME := T#22D22H55M12S817MS;
   S705_LM_DC_2ND_CLAMP6.Error_T1.ATIME := T#22D22H55M13S591MS;
   S705_LM_DC_2ND_CLAMP6.Error_T2.IN := FALSE;
   S705_LM_DC_2ND_CLAMP6.Error_T2.PT := T#4S;
   S705_LM_DC_2ND_CLAMP6.Error_T2.Q := FALSE;
   S705_LM_DC_2ND_CLAMP6.Error_T2.ET := T#0MS;
   S705_LM_DC_2ND_CLAMP6.Error_T2.STATE := B#16#0;
   S705_LM_DC_2ND_CLAMP6.Error_T2.STIME := T#0MS;
   S705_LM_DC_2ND_CLAMP6.Error_T2.ATIME := T#0MS;
   S705_LM_DC_2ND_CLAMP6.CHK_Aux1 := FALSE;
   S705_LM_DC_2ND_CLAMP6.CHK_Aux2 := FALSE;
   S705_LM_DC_2ND_CLAMP6.Error_T1_DN := FALSE;
   S705_LM_DC_2ND_CLAMP6.Error_T2_DN := FALSE;
   S705_LM_DC_2ND_CLAMP6.Adv_Memo := TRUE;
   S705_LM_DC_2ND_CLAMP6.Visu_Adv_Arr[0] := FALSE;
   S705_LM_DC_2ND_CLAMP6.Visu_Adv_Arr[1] := FALSE;
   S705_LM_DC_2ND_CLAMP6.Visu_Adv_Arr[2] := FALSE;
   S705_LM_DC_2ND_CLAMP6.Visu_Adv_Arr[3] := FALSE;
   S705_LM_DC_2ND_CLAMP6.Visu_Adv_Arr[4] := FALSE;
   S705_LM_DC_2ND_CLAMP6.Visu_Adv_Arr[5] := FALSE;
   S705_LM_DC_2ND_CLAMP6.Visu_Adv_Arr[6] := FALSE;
   S705_LM_DC_2ND_CLAMP6.Visu_Adv_Arr[7] := FALSE;
   S705_LM_DC_2ND_CLAMP6.Visu_Adv_Arr[8] := FALSE;
   S705_LM_DC_2ND_CLAMP6.Visu_Adv_Arr[9] := FALSE;
   S705_LM_DC_2ND_CLAMP6.Visu_Adv_Arr[10] := FALSE;
   S705_LM_DC_2ND_CLAMP6.Visu_Adv_Arr[11] := FALSE;
   S705_LM_DC_2ND_CLAMP6.Visu_Adv_Arr[12] := FALSE;
   S705_LM_DC_2ND_CLAMP6.Visu_Adv_Arr[13] := FALSE;
   S705_LM_DC_2ND_CLAMP6.Visu_Adv_Arr[14] := FALSE;
   S705_LM_DC_2ND_CLAMP6.Visu_Adv_Arr[15] := FALSE;
   S705_LM_DC_2ND_CLAMP6.Visu_Ret_Arr[0] := FALSE;
   S705_LM_DC_2ND_CLAMP6.Visu_Ret_Arr[1] := FALSE;
   S705_LM_DC_2ND_CLAMP6.Visu_Ret_Arr[2] := FALSE;
   S705_LM_DC_2ND_CLAMP6.Visu_Ret_Arr[3] := FALSE;
   S705_LM_DC_2ND_CLAMP6.Visu_Ret_Arr[4] := FALSE;
   S705_LM_DC_2ND_CLAMP6.Visu_Ret_Arr[5] := FALSE;
   S705_LM_DC_2ND_CLAMP6.Visu_Ret_Arr[6] := FALSE;
   S705_LM_DC_2ND_CLAMP6.Visu_Ret_Arr[7] := FALSE;
   S705_LM_DC_2ND_CLAMP6.Visu_Ret_Arr[8] := FALSE;
   S705_LM_DC_2ND_CLAMP6.Visu_Ret_Arr[9] := FALSE;
   S705_LM_DC_2ND_CLAMP6.Visu_Ret_Arr[10] := FALSE;
   S705_LM_DC_2ND_CLAMP6.Visu_Ret_Arr[11] := FALSE;
   S705_LM_DC_2ND_CLAMP6.Visu_Ret_Arr[12] := FALSE;
   S705_LM_DC_2ND_CLAMP6.Visu_Ret_Arr[13] := FALSE;
   S705_LM_DC_2ND_CLAMP6.Visu_Ret_Arr[14] := FALSE;
   S705_LM_DC_2ND_CLAMP6.Visu_Ret_Arr[15] := FALSE;
   S705_LM_DC_2ND_CLAMP6.BLK_Move_Ret := 0;
   S705_LM_DC_2ND_CLAMP6.Enable := FALSE;
   S705_LM_DC_2ND_CLAMP6.Adv_End := FALSE;
   S705_LM_DC_2ND_CLAMP6.Ret_End := FALSE;
   S705_LM_DC_2ND_CLAMP7.Enable_Aux := FALSE;
   S705_LM_DC_2ND_CLAMP7.Adv_Amount := 1;
   S705_LM_DC_2ND_CLAMP7.Ret_Amount := 1;
   S705_LM_DC_2ND_CLAMP7.LS_Adv1 := FALSE;
   S705_LM_DC_2ND_CLAMP7.LS_Ret1 := FALSE;
   S705_LM_DC_2ND_CLAMP7.LS_Adv2 := FALSE;
   S705_LM_DC_2ND_CLAMP7.LS_Ret2 := FALSE;
   S705_LM_DC_2ND_CLAMP7.LS_Adv3 := FALSE;
   S705_LM_DC_2ND_CLAMP7.LS_Ret3 := FALSE;
   S705_LM_DC_2ND_CLAMP7.LS_Adv4 := FALSE;
   S705_LM_DC_2ND_CLAMP7.LS_Ret4 := FALSE;
   S705_LM_DC_2ND_CLAMP7.SOL_Adv := FALSE;
   S705_LM_DC_2ND_CLAMP7.SOL_Ret := FALSE;
   S705_LM_DC_2ND_CLAMP7.M_Ready := TRUE;
   S705_LM_DC_2ND_CLAMP7.T_CHK1 := T#4S;
   S705_LM_DC_2ND_CLAMP7.T_CHK2 := T#4S;
   S705_LM_DC_2ND_CLAMP7.PB_Lamp_CHK := FALSE;
   S705_LM_DC_2ND_CLAMP7.PB_Error_Rst := FALSE;
   S705_LM_DC_2ND_CLAMP7.M_FLICK := TRUE;
   S705_LM_DC_2ND_CLAMP7.M_Adv_Err := FALSE;
   S705_LM_DC_2ND_CLAMP7.M_Ret_Err := FALSE;
   S705_LM_DC_2ND_CLAMP7.LP_Adv := FALSE;
   S705_LM_DC_2ND_CLAMP7.LP_Ret := FALSE;
   S705_LM_DC_2ND_CLAMP7.Visu_Adv := W#16#0;
   S705_LM_DC_2ND_CLAMP7.Visu_Ret := W#16#0;
   S705_LM_DC_2ND_CLAMP7.Error_T1.IN := FALSE;
   S705_LM_DC_2ND_CLAMP7.Error_T1.PT := T#4S;
   S705_LM_DC_2ND_CLAMP7.Error_T1.Q := FALSE;
   S705_LM_DC_2ND_CLAMP7.Error_T1.ET := T#0MS;
   S705_LM_DC_2ND_CLAMP7.Error_T1.STATE := B#16#0;
   S705_LM_DC_2ND_CLAMP7.Error_T1.STIME := T#22D22H55M12S817MS;
   S705_LM_DC_2ND_CLAMP7.Error_T1.ATIME := T#22D22H55M13S591MS;
   S705_LM_DC_2ND_CLAMP7.Error_T2.IN := FALSE;
   S705_LM_DC_2ND_CLAMP7.Error_T2.PT := T#4S;
   S705_LM_DC_2ND_CLAMP7.Error_T2.Q := FALSE;
   S705_LM_DC_2ND_CLAMP7.Error_T2.ET := T#0MS;
   S705_LM_DC_2ND_CLAMP7.Error_T2.STATE := B#16#0;
   S705_LM_DC_2ND_CLAMP7.Error_T2.STIME := T#0MS;
   S705_LM_DC_2ND_CLAMP7.Error_T2.ATIME := T#0MS;
   S705_LM_DC_2ND_CLAMP7.CHK_Aux1 := FALSE;
   S705_LM_DC_2ND_CLAMP7.CHK_Aux2 := FALSE;
   S705_LM_DC_2ND_CLAMP7.Error_T1_DN := FALSE;
   S705_LM_DC_2ND_CLAMP7.Error_T2_DN := FALSE;
   S705_LM_DC_2ND_CLAMP7.Adv_Memo := TRUE;
   S705_LM_DC_2ND_CLAMP7.Visu_Adv_Arr[0] := FALSE;
   S705_LM_DC_2ND_CLAMP7.Visu_Adv_Arr[1] := FALSE;
   S705_LM_DC_2ND_CLAMP7.Visu_Adv_Arr[2] := FALSE;
   S705_LM_DC_2ND_CLAMP7.Visu_Adv_Arr[3] := FALSE;
   S705_LM_DC_2ND_CLAMP7.Visu_Adv_Arr[4] := FALSE;
   S705_LM_DC_2ND_CLAMP7.Visu_Adv_Arr[5] := FALSE;
   S705_LM_DC_2ND_CLAMP7.Visu_Adv_Arr[6] := FALSE;
   S705_LM_DC_2ND_CLAMP7.Visu_Adv_Arr[7] := FALSE;
   S705_LM_DC_2ND_CLAMP7.Visu_Adv_Arr[8] := FALSE;
   S705_LM_DC_2ND_CLAMP7.Visu_Adv_Arr[9] := FALSE;
   S705_LM_DC_2ND_CLAMP7.Visu_Adv_Arr[10] := FALSE;
   S705_LM_DC_2ND_CLAMP7.Visu_Adv_Arr[11] := FALSE;
   S705_LM_DC_2ND_CLAMP7.Visu_Adv_Arr[12] := FALSE;
   S705_LM_DC_2ND_CLAMP7.Visu_Adv_Arr[13] := FALSE;
   S705_LM_DC_2ND_CLAMP7.Visu_Adv_Arr[14] := FALSE;
   S705_LM_DC_2ND_CLAMP7.Visu_Adv_Arr[15] := FALSE;
   S705_LM_DC_2ND_CLAMP7.Visu_Ret_Arr[0] := FALSE;
   S705_LM_DC_2ND_CLAMP7.Visu_Ret_Arr[1] := FALSE;
   S705_LM_DC_2ND_CLAMP7.Visu_Ret_Arr[2] := FALSE;
   S705_LM_DC_2ND_CLAMP7.Visu_Ret_Arr[3] := FALSE;
   S705_LM_DC_2ND_CLAMP7.Visu_Ret_Arr[4] := FALSE;
   S705_LM_DC_2ND_CLAMP7.Visu_Ret_Arr[5] := FALSE;
   S705_LM_DC_2ND_CLAMP7.Visu_Ret_Arr[6] := FALSE;
   S705_LM_DC_2ND_CLAMP7.Visu_Ret_Arr[7] := FALSE;
   S705_LM_DC_2ND_CLAMP7.Visu_Ret_Arr[8] := FALSE;
   S705_LM_DC_2ND_CLAMP7.Visu_Ret_Arr[9] := FALSE;
   S705_LM_DC_2ND_CLAMP7.Visu_Ret_Arr[10] := FALSE;
   S705_LM_DC_2ND_CLAMP7.Visu_Ret_Arr[11] := FALSE;
   S705_LM_DC_2ND_CLAMP7.Visu_Ret_Arr[12] := FALSE;
   S705_LM_DC_2ND_CLAMP7.Visu_Ret_Arr[13] := FALSE;
   S705_LM_DC_2ND_CLAMP7.Visu_Ret_Arr[14] := FALSE;
   S705_LM_DC_2ND_CLAMP7.Visu_Ret_Arr[15] := FALSE;
   S705_LM_DC_2ND_CLAMP7.BLK_Move_Ret := 0;
   S705_LM_DC_2ND_CLAMP7.Enable := FALSE;
   S705_LM_DC_2ND_CLAMP7.Adv_End := FALSE;
   S705_LM_DC_2ND_CLAMP7.Ret_End := FALSE;
   S705_LM_DC_1ST_CLAMP5.Enable_Aux := FALSE;
   S705_LM_DC_1ST_CLAMP5.Adv_Amount := 1;
   S705_LM_DC_1ST_CLAMP5.Ret_Amount := 1;
   S705_LM_DC_1ST_CLAMP5.LS_Adv1 := FALSE;
   S705_LM_DC_1ST_CLAMP5.LS_Ret1 := FALSE;
   S705_LM_DC_1ST_CLAMP5.LS_Adv2 := FALSE;
   S705_LM_DC_1ST_CLAMP5.LS_Ret2 := FALSE;
   S705_LM_DC_1ST_CLAMP5.LS_Adv3 := FALSE;
   S705_LM_DC_1ST_CLAMP5.LS_Ret3 := FALSE;
   S705_LM_DC_1ST_CLAMP5.LS_Adv4 := FALSE;
   S705_LM_DC_1ST_CLAMP5.LS_Ret4 := FALSE;
   S705_LM_DC_1ST_CLAMP5.SOL_Adv := FALSE;
   S705_LM_DC_1ST_CLAMP5.SOL_Ret := FALSE;
   S705_LM_DC_1ST_CLAMP5.M_Ready := TRUE;
   S705_LM_DC_1ST_CLAMP5.T_CHK1 := T#4S;
   S705_LM_DC_1ST_CLAMP5.T_CHK2 := T#4S;
   S705_LM_DC_1ST_CLAMP5.PB_Lamp_CHK := FALSE;
   S705_LM_DC_1ST_CLAMP5.PB_Error_Rst := FALSE;
   S705_LM_DC_1ST_CLAMP5.M_FLICK := TRUE;
   S705_LM_DC_1ST_CLAMP5.M_Adv_Err := FALSE;
   S705_LM_DC_1ST_CLAMP5.M_Ret_Err := FALSE;
   S705_LM_DC_1ST_CLAMP5.LP_Adv := FALSE;
   S705_LM_DC_1ST_CLAMP5.LP_Ret := FALSE;
   S705_LM_DC_1ST_CLAMP5.Visu_Adv := W#16#0;
   S705_LM_DC_1ST_CLAMP5.Visu_Ret := W#16#0;
   S705_LM_DC_1ST_CLAMP5.Error_T1.IN := FALSE;
   S705_LM_DC_1ST_CLAMP5.Error_T1.PT := T#4S;
   S705_LM_DC_1ST_CLAMP5.Error_T1.Q := FALSE;
   S705_LM_DC_1ST_CLAMP5.Error_T1.ET := T#0MS;
   S705_LM_DC_1ST_CLAMP5.Error_T1.STATE := B#16#0;
   S705_LM_DC_1ST_CLAMP5.Error_T1.STIME := T#22D22H55M12S68MS;
   S705_LM_DC_1ST_CLAMP5.Error_T1.ATIME := T#22D22H55M12S817MS;
   S705_LM_DC_1ST_CLAMP5.Error_T2.IN := FALSE;
   S705_LM_DC_1ST_CLAMP5.Error_T2.PT := T#4S;
   S705_LM_DC_1ST_CLAMP5.Error_T2.Q := FALSE;
   S705_LM_DC_1ST_CLAMP5.Error_T2.ET := T#0MS;
   S705_LM_DC_1ST_CLAMP5.Error_T2.STATE := B#16#0;
   S705_LM_DC_1ST_CLAMP5.Error_T2.STIME := T#0MS;
   S705_LM_DC_1ST_CLAMP5.Error_T2.ATIME := T#0MS;
   S705_LM_DC_1ST_CLAMP5.CHK_Aux1 := FALSE;
   S705_LM_DC_1ST_CLAMP5.CHK_Aux2 := FALSE;
   S705_LM_DC_1ST_CLAMP5.Error_T1_DN := FALSE;
   S705_LM_DC_1ST_CLAMP5.Error_T2_DN := FALSE;
   S705_LM_DC_1ST_CLAMP5.Adv_Memo := TRUE;
   S705_LM_DC_1ST_CLAMP5.Visu_Adv_Arr[0] := FALSE;
   S705_LM_DC_1ST_CLAMP5.Visu_Adv_Arr[1] := FALSE;
   S705_LM_DC_1ST_CLAMP5.Visu_Adv_Arr[2] := FALSE;
   S705_LM_DC_1ST_CLAMP5.Visu_Adv_Arr[3] := FALSE;
   S705_LM_DC_1ST_CLAMP5.Visu_Adv_Arr[4] := FALSE;
   S705_LM_DC_1ST_CLAMP5.Visu_Adv_Arr[5] := FALSE;
   S705_LM_DC_1ST_CLAMP5.Visu_Adv_Arr[6] := FALSE;
   S705_LM_DC_1ST_CLAMP5.Visu_Adv_Arr[7] := FALSE;
   S705_LM_DC_1ST_CLAMP5.Visu_Adv_Arr[8] := FALSE;
   S705_LM_DC_1ST_CLAMP5.Visu_Adv_Arr[9] := FALSE;
   S705_LM_DC_1ST_CLAMP5.Visu_Adv_Arr[10] := FALSE;
   S705_LM_DC_1ST_CLAMP5.Visu_Adv_Arr[11] := FALSE;
   S705_LM_DC_1ST_CLAMP5.Visu_Adv_Arr[12] := FALSE;
   S705_LM_DC_1ST_CLAMP5.Visu_Adv_Arr[13] := FALSE;
   S705_LM_DC_1ST_CLAMP5.Visu_Adv_Arr[14] := FALSE;
   S705_LM_DC_1ST_CLAMP5.Visu_Adv_Arr[15] := FALSE;
   S705_LM_DC_1ST_CLAMP5.Visu_Ret_Arr[0] := FALSE;
   S705_LM_DC_1ST_CLAMP5.Visu_Ret_Arr[1] := FALSE;
   S705_LM_DC_1ST_CLAMP5.Visu_Ret_Arr[2] := FALSE;
   S705_LM_DC_1ST_CLAMP5.Visu_Ret_Arr[3] := FALSE;
   S705_LM_DC_1ST_CLAMP5.Visu_Ret_Arr[4] := FALSE;
   S705_LM_DC_1ST_CLAMP5.Visu_Ret_Arr[5] := FALSE;
   S705_LM_DC_1ST_CLAMP5.Visu_Ret_Arr[6] := FALSE;
   S705_LM_DC_1ST_CLAMP5.Visu_Ret_Arr[7] := FALSE;
   S705_LM_DC_1ST_CLAMP5.Visu_Ret_Arr[8] := FALSE;
   S705_LM_DC_1ST_CLAMP5.Visu_Ret_Arr[9] := FALSE;
   S705_LM_DC_1ST_CLAMP5.Visu_Ret_Arr[10] := FALSE;
   S705_LM_DC_1ST_CLAMP5.Visu_Ret_Arr[11] := FALSE;
   S705_LM_DC_1ST_CLAMP5.Visu_Ret_Arr[12] := FALSE;
   S705_LM_DC_1ST_CLAMP5.Visu_Ret_Arr[13] := FALSE;
   S705_LM_DC_1ST_CLAMP5.Visu_Ret_Arr[14] := FALSE;
   S705_LM_DC_1ST_CLAMP5.Visu_Ret_Arr[15] := FALSE;
   S705_LM_DC_1ST_CLAMP5.BLK_Move_Ret := 0;
   S705_LM_DC_1ST_CLAMP5.Enable := FALSE;
   S705_LM_DC_1ST_CLAMP5.Adv_End := FALSE;
   S705_LM_DC_1ST_CLAMP5.Ret_End := FALSE;
END_DATA_BLOCK

FUNCTION FC 113 : VOID
TITLE =
NAME : DAECHA
VERSION : 0.1

BEGIN
NETWORK
TITLE =
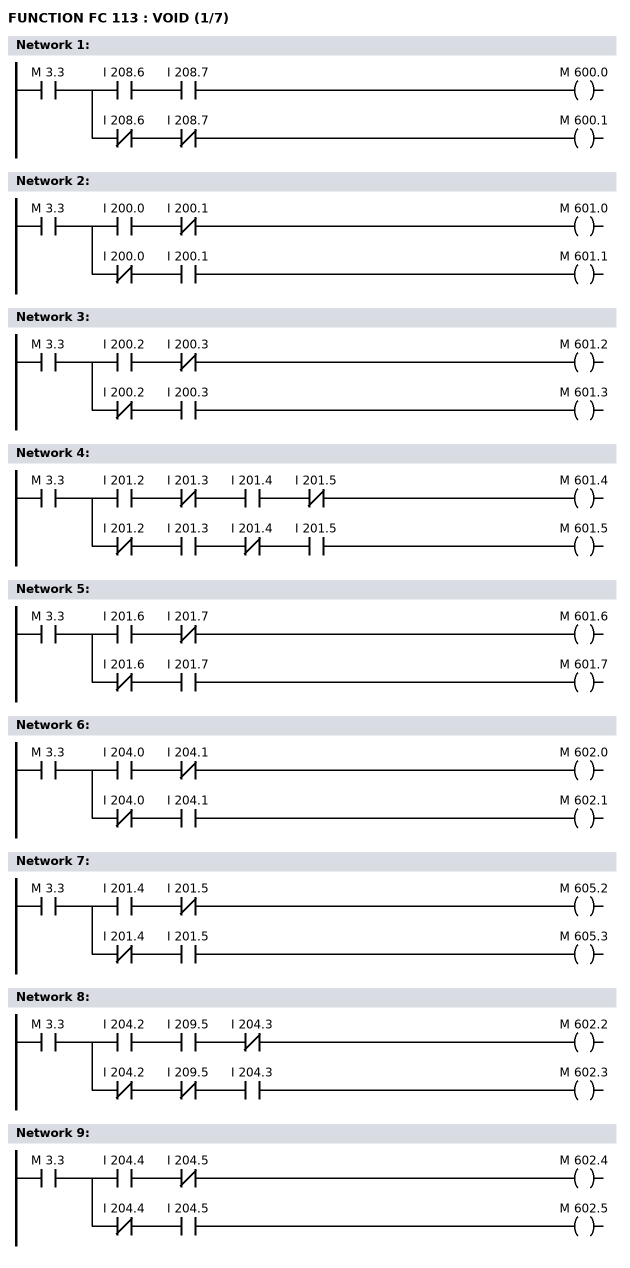

      A     M      3.3;
      =     L      0.0;
      A     L      0.0;
      A     I    208.6;
      A     I    208.7;
      =     M    600.0;
      A     L      0.0;
      AN    I    208.6;
      AN    I    208.7;
      =     M    600.1;
NETWORK
TITLE =

      A     M      3.3;
      =     L      0.0;
      A     L      0.0;
      A     I    200.0;
      AN    I    200.1;
      =     M    601.0;
      A     L      0.0;
      AN    I    200.0;
      A     I    200.1;
      =     M    601.1;
NETWORK
TITLE =

      A     M      3.3;
      =     L      0.0;
      A     L      0.0;
      A     I    200.2;
      AN    I    200.3;
      =     M    601.2;
      A     L      0.0;
      AN    I    200.2;
      A     I    200.3;
      =     M    601.3;
NETWORK
TITLE =

      A     M      3.3;
      =     L      0.0;
      A     L      0.0;
      A     I    201.2;
      AN    I    201.3;
      A     I    201.4;
      AN    I    201.5;
      =     M    601.4;
      A     L      0.0;
      AN    I    201.2;
      A     I    201.3;
      AN    I    201.4;
      A     I    201.5;
      =     M    601.5;
NETWORK
TITLE =

      A     M      3.3;
      =     L      0.0;
      A     L      0.0;
      A     I    201.6;
      AN    I    201.7;
      =     M    601.6;
      A     L      0.0;
      AN    I    201.6;
      A     I    201.7;
      =     M    601.7;
NETWORK
TITLE =

      A     M      3.3;
      =     L      0.0;
      A     L      0.0;
      A     I    204.0;
      AN    I    204.1;
      =     M    602.0;
      A     L      0.0;
      AN    I    204.0;
      A     I    204.1;
      =     M    602.1;
NETWORK
TITLE =

      A     M      3.3;
      =     L      0.0;
      A     L      0.0;
      A     I    201.4;
      AN    I    201.5;
      =     M    605.2;
      A     L      0.0;
      AN    I    201.4;
      A     I    201.5;
      =     M    605.3;
NETWORK
TITLE =

      A     M      3.3;
      =     L      0.0;
      A     L      0.0;
      A     I    204.2;
      A     I    209.5;
      AN    I    204.3;
      =     M    602.2;
      A     L      0.0;
      AN    I    204.2;
      AN    I    209.5;
      A     I    204.3;
      =     M    602.3;
NETWORK
TITLE =

      A     M      3.3;
      =     L      0.0;
      A     L      0.0;
      A     I    204.4;
      AN    I    204.5;
      =     M    602.4;
      A     L      0.0;
      AN    I    204.4;
      A     I    204.5;
      =     M    602.5;
NETWORK
TITLE =
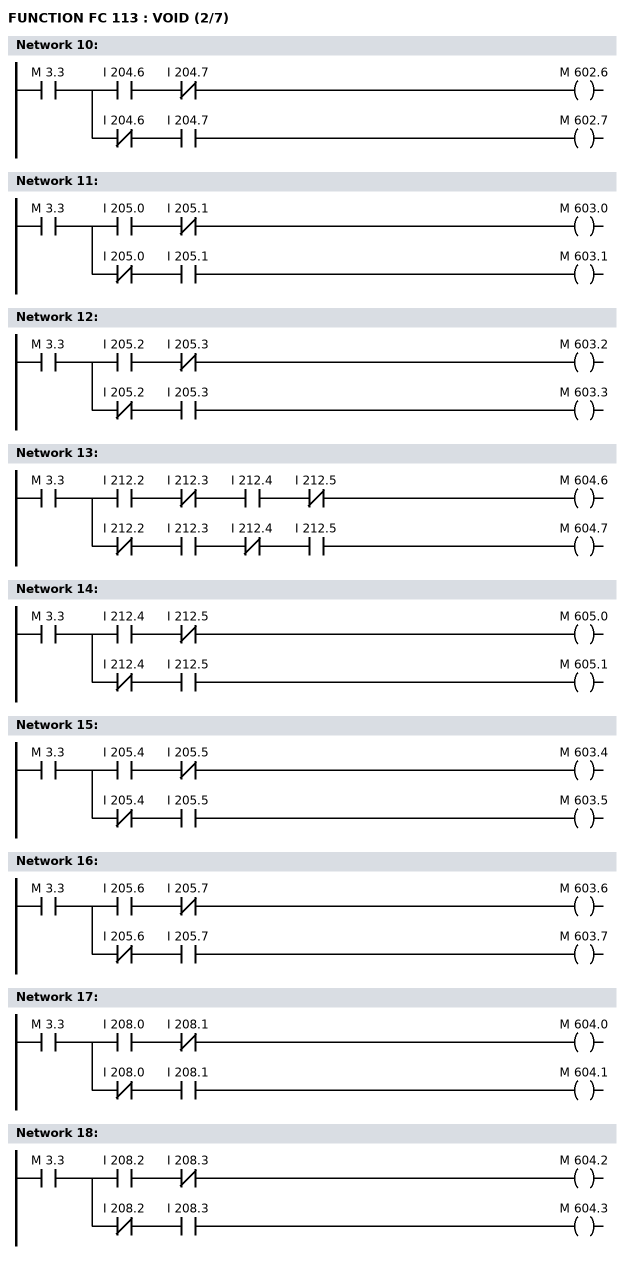

      A     M      3.3;
      =     L      0.0;
      A     L      0.0;
      A     I    204.6;
      AN    I    204.7;
      =     M    602.6;
      A     L      0.0;
      AN    I    204.6;
      A     I    204.7;
      =     M    602.7;
NETWORK
TITLE =

      A     M      3.3;
      =     L      0.0;
      A     L      0.0;
      A     I    205.0;
      AN    I    205.1;
      =     M    603.0;
      A     L      0.0;
      AN    I    205.0;
      A     I    205.1;
      =     M    603.1;
NETWORK
TITLE =

      A     M      3.3;
      =     L      0.0;
      A     L      0.0;
      A     I    205.2;
      AN    I    205.3;
      =     M    603.2;
      A     L      0.0;
      AN    I    205.2;
      A     I    205.3;
      =     M    603.3;
NETWORK
TITLE =

      A     M      3.3;
      =     L      0.0;
      A     L      0.0;
      A     I    212.2;
      AN    I    212.3;
      A     I    212.4;
      AN    I    212.5;
      =     M    604.6;
      A     L      0.0;
      AN    I    212.2;
      A     I    212.3;
      AN    I    212.4;
      A     I    212.5;
      =     M    604.7;
NETWORK
TITLE =

      A     M      3.3;
      =     L      0.0;
      A     L      0.0;
      A     I    212.4;
      AN    I    212.5;
      =     M    605.0;
      A     L      0.0;
      AN    I    212.4;
      A     I    212.5;
      =     M    605.1;
NETWORK
TITLE =

      A     M      3.3;
      =     L      0.0;
      A     L      0.0;
      A     I    205.4;
      AN    I    205.5;
      =     M    603.4;
      A     L      0.0;
      AN    I    205.4;
      A     I    205.5;
      =     M    603.5;
NETWORK
TITLE =

      A     M      3.3;
      =     L      0.0;
      A     L      0.0;
      A     I    205.6;
      AN    I    205.7;
      =     M    603.6;
      A     L      0.0;
      AN    I    205.6;
      A     I    205.7;
      =     M    603.7;
NETWORK
TITLE =

      A     M      3.3;
      =     L      0.0;
      A     L      0.0;
      A     I    208.0;
      AN    I    208.1;
      =     M    604.0;
      A     L      0.0;
      AN    I    208.0;
      A     I    208.1;
      =     M    604.1;
NETWORK
TITLE =

      A     M      3.3;
      =     L      0.0;
      A     L      0.0;
      A     I    208.2;
      AN    I    208.3;
      =     M    604.2;
      A     L      0.0;
      AN    I    208.2;
      A     I    208.3;
      =     M    604.3;
NETWORK
TITLE =
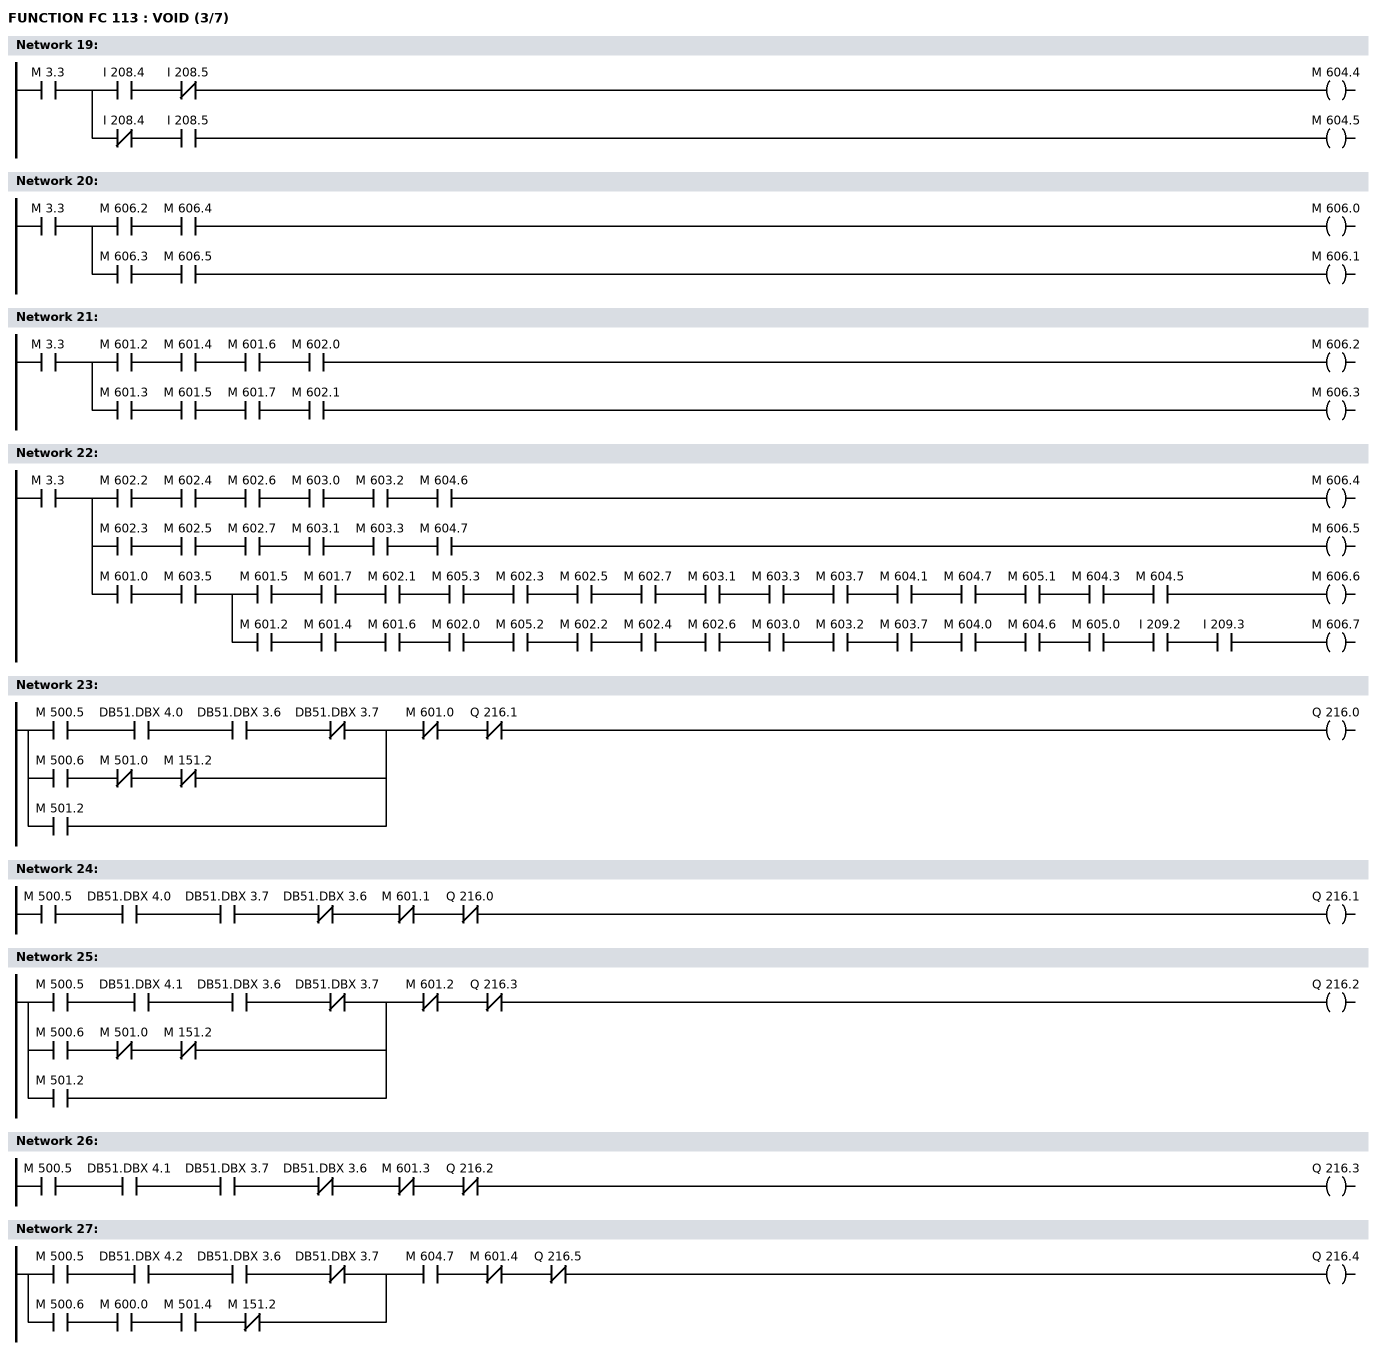

      A     M      3.3;
      =     L      0.0;
      A     L      0.0;
      A     I    208.4;
      AN    I    208.5;
      =     M    604.4;
      A     L      0.0;
      AN    I    208.4;
      A     I    208.5;
      =     M    604.5;
NETWORK
TITLE =

      A     M      3.3;
      =     L      0.0;
      A     L      0.0;
      A     M    606.2;
      A     M    606.4;
      =     M    606.0;
      A     L      0.0;
      A     M    606.3;
      A     M    606.5;
      =     M    606.1;
NETWORK
TITLE =

      A     M      3.3;
      =     L      0.0;
      A     L      0.0;
      A     M    601.2;
      A     M    601.4;
      A     M    601.6;
      A     M    602.0;
      =     M    606.2;
      A     L      0.0;
      A     M    601.3;
      A     M    601.5;
      A     M    601.7;
      A     M    602.1;
      =     M    606.3;
NETWORK
TITLE =

      A     M      3.3;
      =     L      0.0;
      A     L      0.0;
      A     M    602.2;
      A     M    602.4;
      A     M    602.6;
      A     M    603.0;
      A     M    603.2;
      A     M    604.6;
      =     M    606.4;
      A     L      0.0;
      A     M    602.3;
      A     M    602.5;
      A     M    602.7;
      A     M    603.1;
      A     M    603.3;
      A     M    604.7;
      =     M    606.5;
      A     L      0.0;
      A     M    601.0;
      A     M    603.5;
      =     L      0.1;
      A     L      0.1;
      A     M    601.5;
      A     M    601.7;
      A     M    602.1;
      A     M    605.3;
      A     M    602.3;
      A     M    602.5;
      A     M    602.7;
      A     M    603.1;
      A     M    603.3;
      A     M    603.7;
      A     M    604.1;
      A     M    604.7;
      A     M    605.1;
      A     M    604.3;
      A     M    604.5;
      =     M    606.6;
      A     L      0.1;
      A     M    601.2;
      A     M    601.4;
      A     M    601.6;
      A     M    602.0;
      A     M    605.2;
      A     M    602.2;
      A     M    602.4;
      A     M    602.6;
      A     M    603.0;
      A     M    603.2;
      A     M    603.7;
      A     M    604.0;
      A     M    604.6;
      A     M    605.0;
      A     I    209.2;
      A     I    209.3;
      =     M    606.7;
NETWORK
TITLE =

      A(    ;
      A     M    500.5;
      A     DB51.DBX    4.0;
      A     DB51.DBX    3.6;
      AN    DB51.DBX    3.7;
      O     ;
      A     M    500.6;
      AN    M    501.0;
      AN    M    151.2;
      O     M    501.2;
      )     ;
      AN    M    601.0;
      AN    Q    216.1;
      =     Q    216.0;
NETWORK
TITLE =

      A     M    500.5;
      A     DB51.DBX    4.0;
      A     DB51.DBX    3.7;
      AN    DB51.DBX    3.6;
      AN    M    601.1;
      AN    Q    216.0;
      =     Q    216.1;
NETWORK
TITLE =

      A(    ;
      A     M    500.5;
      A     DB51.DBX    4.1;
      A     DB51.DBX    3.6;
      AN    DB51.DBX    3.7;
      O     ;
      A     M    500.6;
      AN    M    501.0;
      AN    M    151.2;
      O     M    501.2;
      )     ;
      AN    M    601.2;
      AN    Q    216.3;
      =     Q    216.2;
NETWORK
TITLE =

      A     M    500.5;
      A     DB51.DBX    4.1;
      A     DB51.DBX    3.7;
      AN    DB51.DBX    3.6;
      AN    M    601.3;
      AN    Q    216.2;
      =     Q    216.3;
NETWORK
TITLE =

      A(    ;
      A     M    500.5;
      A     DB51.DBX    4.2;
      A     DB51.DBX    3.6;
      AN    DB51.DBX    3.7;
      O     ;
      A     M    500.6;
      A     M    600.0;
      A     M    501.4;
      AN    M    151.2;
      )     ;
      A     M    604.7;
      AN    M    601.4;
      AN    Q    216.5;
      =     Q    216.4;
NETWORK
TITLE =
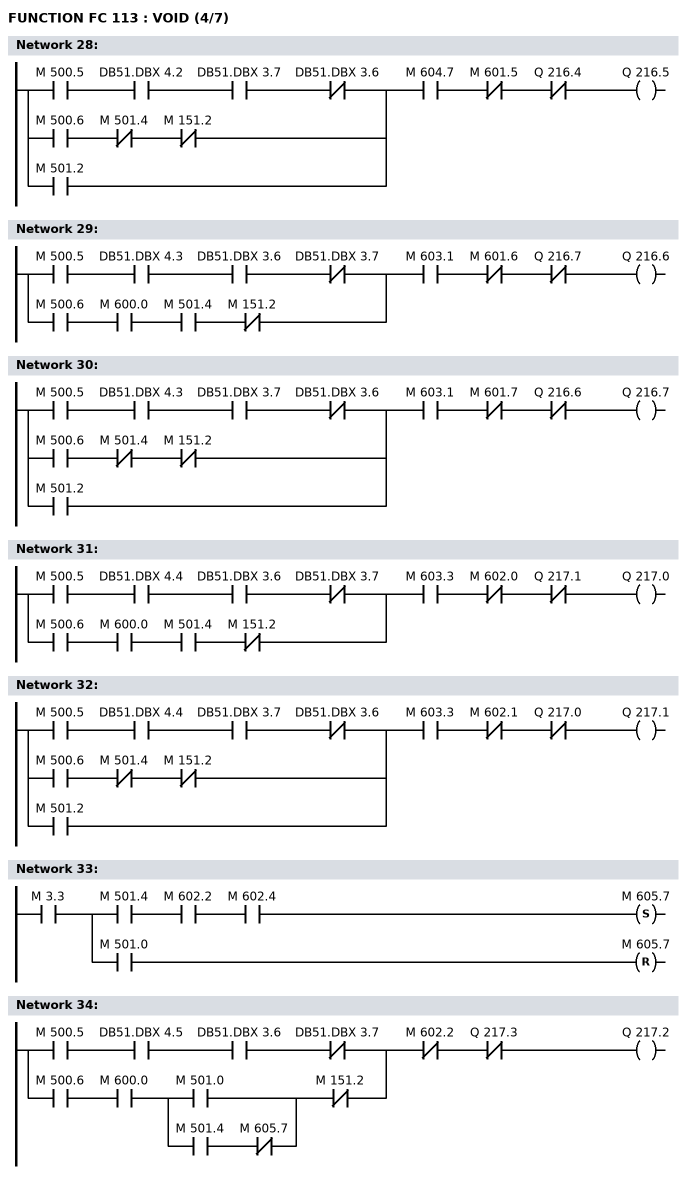

      A(    ;
      A     M    500.5;
      A     DB51.DBX    4.2;
      A     DB51.DBX    3.7;
      AN    DB51.DBX    3.6;
      O     ;
      A     M    500.6;
      AN    M    501.4;
      AN    M    151.2;
      O     M    501.2;
      )     ;
      A     M    604.7;
      AN    M    601.5;
      AN    Q    216.4;
      =     Q    216.5;
NETWORK
TITLE =

      A(    ;
      A     M    500.5;
      A     DB51.DBX    4.3;
      A     DB51.DBX    3.6;
      AN    DB51.DBX    3.7;
      O     ;
      A     M    500.6;
      A     M    600.0;
      A     M    501.4;
      AN    M    151.2;
      )     ;
      A     M    603.1;
      AN    M    601.6;
      AN    Q    216.7;
      =     Q    216.6;
NETWORK
TITLE =

      A(    ;
      A     M    500.5;
      A     DB51.DBX    4.3;
      A     DB51.DBX    3.7;
      AN    DB51.DBX    3.6;
      O     ;
      A     M    500.6;
      AN    M    501.4;
      AN    M    151.2;
      O     M    501.2;
      )     ;
      A     M    603.1;
      AN    M    601.7;
      AN    Q    216.6;
      =     Q    216.7;
NETWORK
TITLE =

      A(    ;
      A     M    500.5;
      A     DB51.DBX    4.4;
      A     DB51.DBX    3.6;
      AN    DB51.DBX    3.7;
      O     ;
      A     M    500.6;
      A     M    600.0;
      A     M    501.4;
      AN    M    151.2;
      )     ;
      A     M    603.3;
      AN    M    602.0;
      AN    Q    217.1;
      =     Q    217.0;
NETWORK
TITLE =

      A(    ;
      A     M    500.5;
      A     DB51.DBX    4.4;
      A     DB51.DBX    3.7;
      AN    DB51.DBX    3.6;
      O     ;
      A     M    500.6;
      AN    M    501.4;
      AN    M    151.2;
      O     M    501.2;
      )     ;
      A     M    603.3;
      AN    M    602.1;
      AN    Q    217.0;
      =     Q    217.1;
NETWORK
TITLE =

      A     M      3.3;
      =     L      0.0;
      A     L      0.0;
      A     M    501.4;
      A     M    602.2;
      A     M    602.4;
      S     M    605.7;
      A     L      0.0;
      A     M    501.0;
      R     M    605.7;
NETWORK
TITLE =

      A(    ;
      A     M    500.5;
      A     DB51.DBX    4.5;
      A     DB51.DBX    3.6;
      AN    DB51.DBX    3.7;
      O     ;
      A     M    500.6;
      A     M    600.0;
      A(    ;
      O     M    501.0;
      O     ;
      A     M    501.4;
      AN    M    605.7;
      )     ;
      AN    M    151.2;
      )     ;
      AN    M    602.2;
      AN    Q    217.3;
      =     Q    217.2;
NETWORK
TITLE =
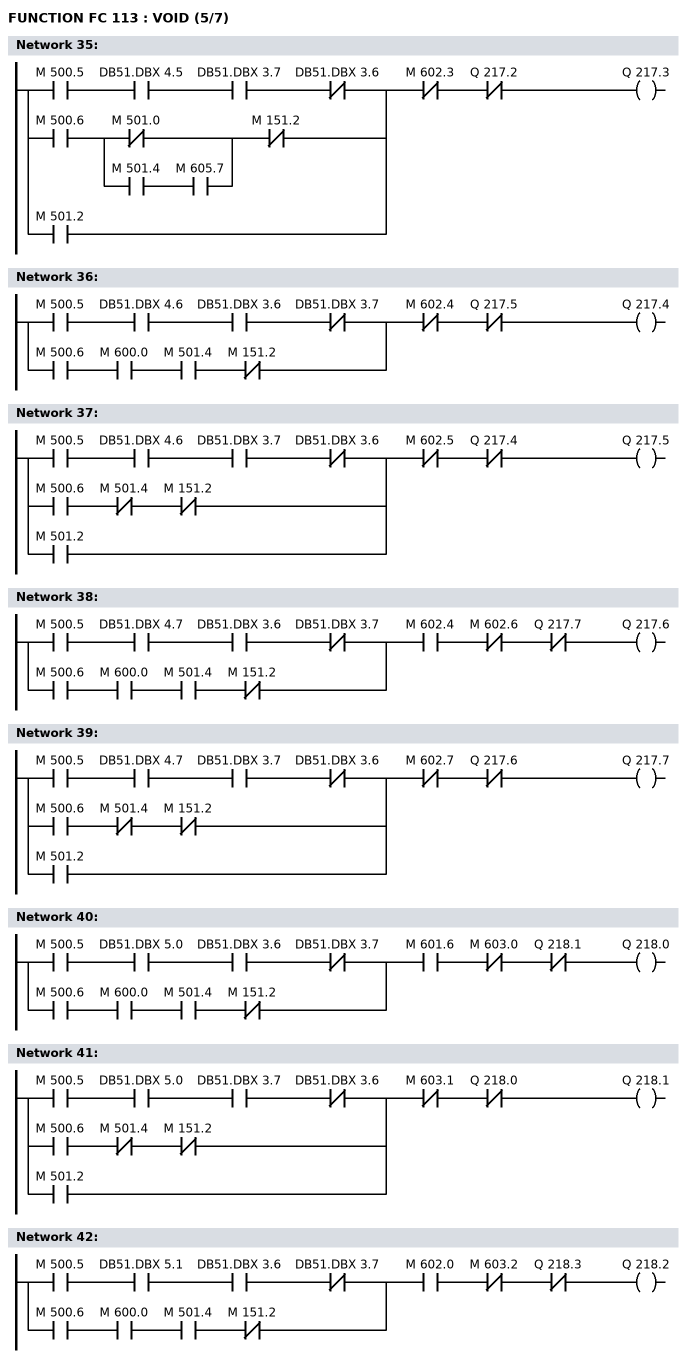

      A(    ;
      A     M    500.5;
      A     DB51.DBX    4.5;
      A     DB51.DBX    3.7;
      AN    DB51.DBX    3.6;
      O     ;
      A     M    500.6;
      A(    ;
      ON    M    501.0;
      O     ;
      A     M    501.4;
      A     M    605.7;
      )     ;
      AN    M    151.2;
      O     M    501.2;
      )     ;
      AN    M    602.3;
      AN    Q    217.2;
      =     Q    217.3;
NETWORK
TITLE =

      A(    ;
      A     M    500.5;
      A     DB51.DBX    4.6;
      A     DB51.DBX    3.6;
      AN    DB51.DBX    3.7;
      O     ;
      A     M    500.6;
      A     M    600.0;
      A     M    501.4;
      AN    M    151.2;
      )     ;
      AN    M    602.4;
      AN    Q    217.5;
      =     Q    217.4;
NETWORK
TITLE =

      A(    ;
      A     M    500.5;
      A     DB51.DBX    4.6;
      A     DB51.DBX    3.7;
      AN    DB51.DBX    3.6;
      O     ;
      A     M    500.6;
      AN    M    501.4;
      AN    M    151.2;
      O     M    501.2;
      )     ;
      AN    M    602.5;
      AN    Q    217.4;
      =     Q    217.5;
NETWORK
TITLE =

      A(    ;
      A     M    500.5;
      A     DB51.DBX    4.7;
      A     DB51.DBX    3.6;
      AN    DB51.DBX    3.7;
      O     ;
      A     M    500.6;
      A     M    600.0;
      A     M    501.4;
      AN    M    151.2;
      )     ;
      A     M    602.4;
      AN    M    602.6;
      AN    Q    217.7;
      =     Q    217.6;
NETWORK
TITLE =

      A(    ;
      A     M    500.5;
      A     DB51.DBX    4.7;
      A     DB51.DBX    3.7;
      AN    DB51.DBX    3.6;
      O     ;
      A     M    500.6;
      AN    M    501.4;
      AN    M    151.2;
      O     M    501.2;
      )     ;
      AN    M    602.7;
      AN    Q    217.6;
      =     Q    217.7;
NETWORK
TITLE =

      A(    ;
      A     M    500.5;
      A     DB51.DBX    5.0;
      A     DB51.DBX    3.6;
      AN    DB51.DBX    3.7;
      O     ;
      A     M    500.6;
      A     M    600.0;
      A     M    501.4;
      AN    M    151.2;
      )     ;
      A     M    601.6;
      AN    M    603.0;
      AN    Q    218.1;
      =     Q    218.0;
NETWORK
TITLE =

      A(    ;
      A     M    500.5;
      A     DB51.DBX    5.0;
      A     DB51.DBX    3.7;
      AN    DB51.DBX    3.6;
      O     ;
      A     M    500.6;
      AN    M    501.4;
      AN    M    151.2;
      O     M    501.2;
      )     ;
      AN    M    603.1;
      AN    Q    218.0;
      =     Q    218.1;
NETWORK
TITLE =

      A(    ;
      A     M    500.5;
      A     DB51.DBX    5.1;
      A     DB51.DBX    3.6;
      AN    DB51.DBX    3.7;
      O     ;
      A     M    500.6;
      A     M    600.0;
      A     M    501.4;
      AN    M    151.2;
      )     ;
      A     M    602.0;
      AN    M    603.2;
      AN    Q    218.3;
      =     Q    218.2;
NETWORK
TITLE =
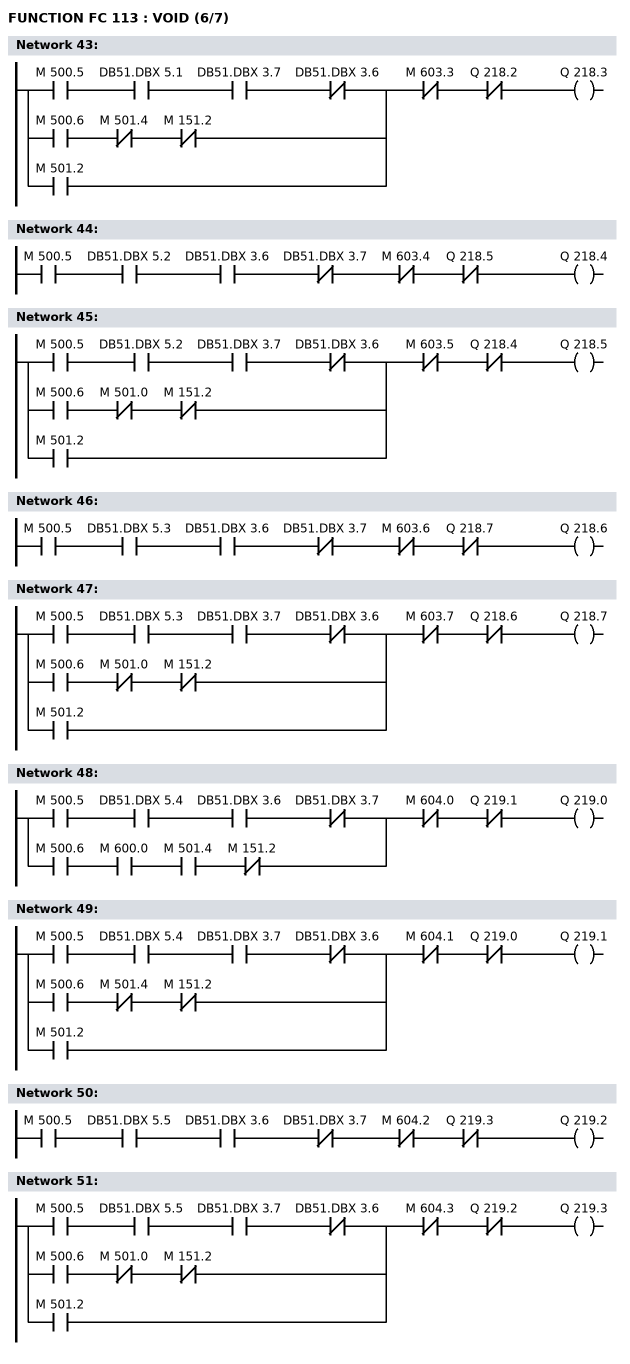

      A(    ;
      A     M    500.5;
      A     DB51.DBX    5.1;
      A     DB51.DBX    3.7;
      AN    DB51.DBX    3.6;
      O     ;
      A     M    500.6;
      AN    M    501.4;
      AN    M    151.2;
      O     M    501.2;
      )     ;
      AN    M    603.3;
      AN    Q    218.2;
      =     Q    218.3;
NETWORK
TITLE =

      A     M    500.5;
      A     DB51.DBX    5.2;
      A     DB51.DBX    3.6;
      AN    DB51.DBX    3.7;
      AN    M    603.4;
      AN    Q    218.5;
      =     Q    218.4;
NETWORK
TITLE =

      A(    ;
      A     M    500.5;
      A     DB51.DBX    5.2;
      A     DB51.DBX    3.7;
      AN    DB51.DBX    3.6;
      O     ;
      A     M    500.6;
      AN    M    501.0;
      AN    M    151.2;
      O     M    501.2;
      )     ;
      AN    M    603.5;
      AN    Q    218.4;
      =     Q    218.5;
NETWORK
TITLE =

      A     M    500.5;
      A     DB51.DBX    5.3;
      A     DB51.DBX    3.6;
      AN    DB51.DBX    3.7;
      AN    M    603.6;
      AN    Q    218.7;
      =     Q    218.6;
NETWORK
TITLE =

      A(    ;
      A     M    500.5;
      A     DB51.DBX    5.3;
      A     DB51.DBX    3.7;
      AN    DB51.DBX    3.6;
      O     ;
      A     M    500.6;
      AN    M    501.0;
      AN    M    151.2;
      O     M    501.2;
      )     ;
      AN    M    603.7;
      AN    Q    218.6;
      =     Q    218.7;
NETWORK
TITLE =

      A(    ;
      A     M    500.5;
      A     DB51.DBX    5.4;
      A     DB51.DBX    3.6;
      AN    DB51.DBX    3.7;
      O     ;
      A     M    500.6;
      A     M    600.0;
      A     M    501.4;
      AN    M    151.2;
      )     ;
      AN    M    604.0;
      AN    Q    219.1;
      =     Q    219.0;
NETWORK
TITLE =

      A(    ;
      A     M    500.5;
      A     DB51.DBX    5.4;
      A     DB51.DBX    3.7;
      AN    DB51.DBX    3.6;
      O     ;
      A     M    500.6;
      AN    M    501.4;
      AN    M    151.2;
      O     M    501.2;
      )     ;
      AN    M    604.1;
      AN    Q    219.0;
      =     Q    219.1;
NETWORK
TITLE =

      A     M    500.5;
      A     DB51.DBX    5.5;
      A     DB51.DBX    3.6;
      AN    DB51.DBX    3.7;
      AN    M    604.2;
      AN    Q    219.3;
      =     Q    219.2;
NETWORK
TITLE =

      A(    ;
      A     M    500.5;
      A     DB51.DBX    5.5;
      A     DB51.DBX    3.7;
      AN    DB51.DBX    3.6;
      O     ;
      A     M    500.6;
      AN    M    501.0;
      AN    M    151.2;
      O     M    501.2;
      )     ;
      AN    M    604.3;
      AN    Q    219.2;
      =     Q    219.3;
NETWORK
TITLE =
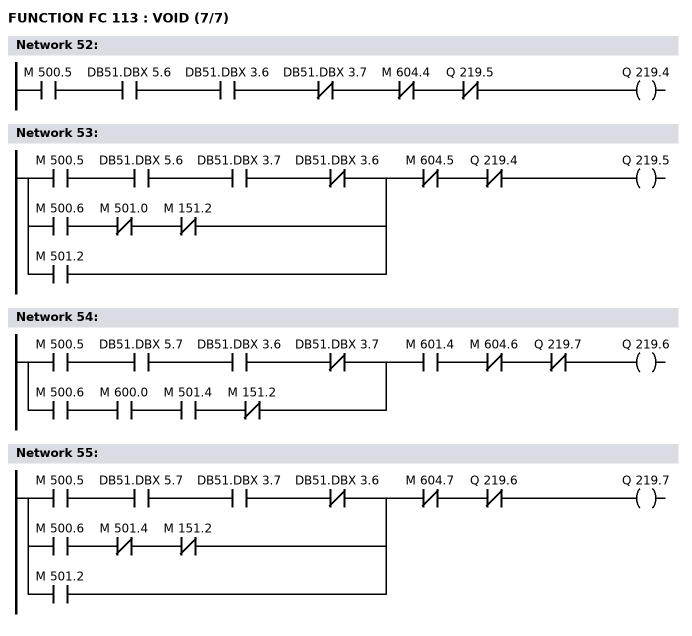

      A     M    500.5;
      A     DB51.DBX    5.6;
      A     DB51.DBX    3.6;
      AN    DB51.DBX    3.7;
      AN    M    604.4;
      AN    Q    219.5;
      =     Q    219.4;
NETWORK
TITLE =

      A(    ;
      A     M    500.5;
      A     DB51.DBX    5.6;
      A     DB51.DBX    3.7;
      AN    DB51.DBX    3.6;
      O     ;
      A     M    500.6;
      AN    M    501.0;
      AN    M    151.2;
      O     M    501.2;
      )     ;
      AN    M    604.5;
      AN    Q    219.4;
      =     Q    219.5;
NETWORK
TITLE =

      A(    ;
      A     M    500.5;
      A     DB51.DBX    5.7;
      A     DB51.DBX    3.6;
      AN    DB51.DBX    3.7;
      O     ;
      A     M    500.6;
      A     M    600.0;
      A     M    501.4;
      AN    M    151.2;
      )     ;
      A     M    601.4;
      AN    M    604.6;
      AN    Q    219.7;
      =     Q    219.6;
NETWORK
TITLE =

      A(    ;
      A     M    500.5;
      A     DB51.DBX    5.7;
      A     DB51.DBX    3.7;
      AN    DB51.DBX    3.6;
      O     ;
      A     M    500.6;
      AN    M    501.4;
      AN    M    151.2;
      O     M    501.2;
      )     ;
      AN    M    604.7;
      AN    Q    219.6;
      =     Q    219.7;
END_FUNCTION

FUNCTION_BLOCK FB 114
TITLE =
VERSION : 0.1


VAR
  S705_TL_DC_PIN : FB 426;
  S705_TL_DC_LATCH1 : FB 426;
  S705_TL_DC_LATCH2 : FB 426;
  S705_TL_DC_1ST_CLAMP1 : FB 426;
  S705_TL_DC_1ST_CLAMP2 : FB 426;
  S705_TL_DC_1ST_CLAMP3 : FB 426;
  S705_TL_DC_2ND_CLAMP1 : FB 426;
  S705_TL_DC_2ND_CLAMP2 : FB 426;
  S705_TL_DC_U261 : FB 426;
  S705_TL_DC_U261_CLAMP : FB 426;
  S705_TL_DC_U269 : FB 426;
  S705_TL_DC_U269_CLAMP : FB 426;
  S705_TL_DC_3RD_CLAMP : FB 426;
  S705_TL_DC_U262_1_UP_DN : FB 426;
  S705_TL_DC_U262_1 : FB 426;
  S705_TL_DC_U262_1_CLAMP : FB 426;
  S705_TL_DC_U261_2_CLAMP : FB 426;
END_VAR
BEGIN
NETWORK
TITLE =
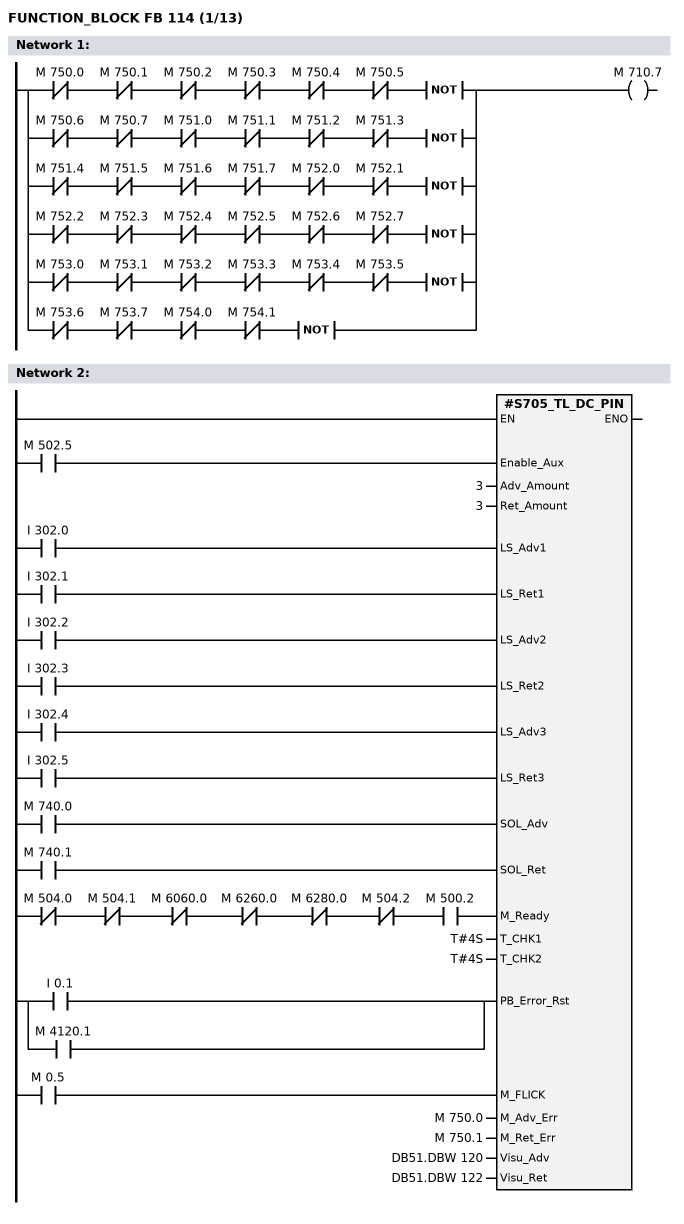

      AN    M    750.0;
      AN    M    750.1;
      AN    M    750.2;
      AN    M    750.3;
      AN    M    750.4;
      AN    M    750.5;
      NOT   ;
      O(    ;
      AN    M    750.6;
      AN    M    750.7;
      AN    M    751.0;
      AN    M    751.1;
      AN    M    751.2;
      AN    M    751.3;
      NOT   ;
      )     ;
      O(    ;
      AN    M    751.4;
      AN    M    751.5;
      AN    M    751.6;
      AN    M    751.7;
      AN    M    752.0;
      AN    M    752.1;
      NOT   ;
      )     ;
      O(    ;
      AN    M    752.2;
      AN    M    752.3;
      AN    M    752.4;
      AN    M    752.5;
      AN    M    752.6;
      AN    M    752.7;
      NOT   ;
      )     ;
      O(    ;
      AN    M    753.0;
      AN    M    753.1;
      AN    M    753.2;
      AN    M    753.3;
      AN    M    753.4;
      AN    M    753.5;
      NOT   ;
      )     ;
      O(    ;
      AN    M    753.6;
      AN    M    753.7;
      AN    M    754.0;
      AN    M    754.1;
      NOT   ;
      )     ;
      =     M    710.7;
NETWORK
TITLE =

      A     M    502.5;
      =     L      0.0;
      BLD   103;
      A     I    302.0;
      =     L      0.1;
      BLD   103;
      A     I    302.1;
      =     L      0.2;
      BLD   103;
      A     I    302.2;
      =     L      0.3;
      BLD   103;
      A     I    302.3;
      =     L      0.4;
      BLD   103;
      A     I    302.4;
      =     L      0.5;
      BLD   103;
      A     I    302.5;
      =     L      0.6;
      BLD   103;
      A     M    740.0;
      =     L      2.1;
      BLD   103;
      A     M    740.1;
      =     L      2.2;
      BLD   103;
      AN    M    504.0;
      AN    M    504.1;
      AN    M   6060.0;
      AN    M   6260.0;
      AN    M   6280.0;
      AN    M    504.2;
      A     M    500.2;
      =     L      2.3;
      BLD   103;
      A(    ;
      O     I      0.1;
      O     M   4120.1;
      )     ;
      =     L      2.5;
      BLD   103;
      A     M      0.5;
      =     L      2.6;
      BLD   103;
      CALL #S705_TL_DC_PIN (
           Enable_Aux               := L      0.0,
           Adv_Amount               := 3,
           Ret_Amount               := 3,
           LS_Adv1                  := L      0.1,
           LS_Ret1                  := L      0.2,
           LS_Adv2                  := L      0.3,
           LS_Ret2                  := L      0.4,
           LS_Adv3                  := L      0.5,
           LS_Ret3                  := L      0.6,
           SOL_Adv                  := L      2.1,
           SOL_Ret                  := L      2.2,
           M_Ready                  := L      2.3,
           T_CHK1                   := T#4S,
           T_CHK2                   := T#4S,
           PB_Error_Rst             := L      2.5,
           M_FLICK                  := L      2.6,
           M_Adv_Err                := M    750.0,
           M_Ret_Err                := M    750.1,
           Visu_Adv                 := DB51.DBW  120,
           Visu_Ret                 := DB51.DBW  122);
      NOP   0;
NETWORK
TITLE =
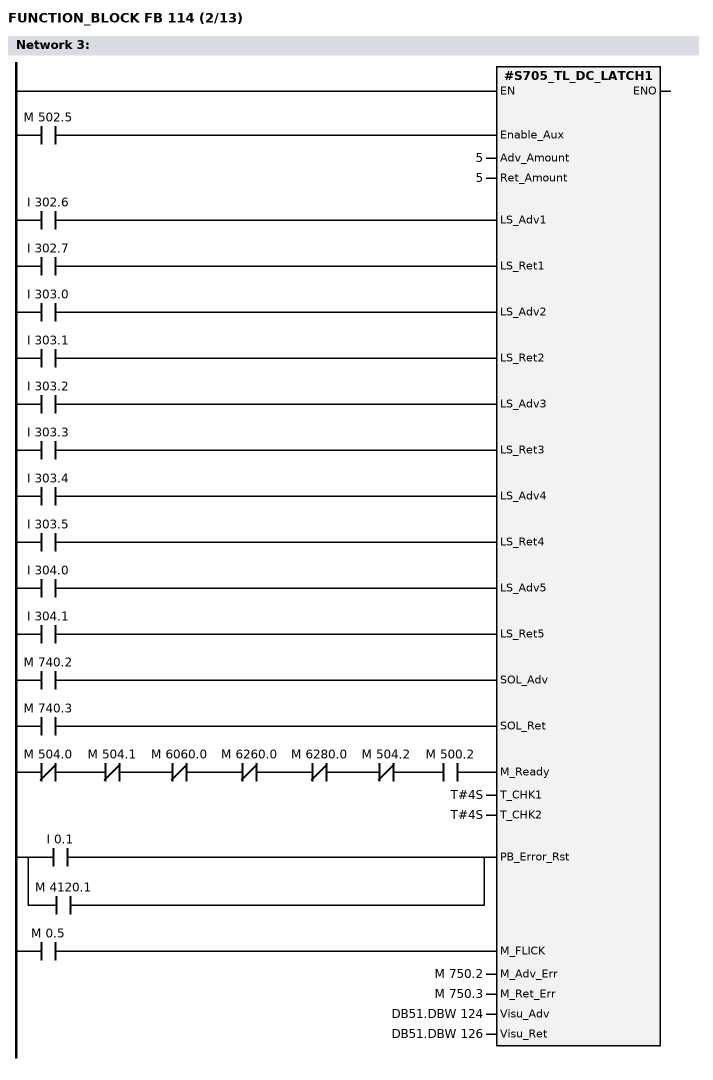

      A     M    502.5;
      =     L      0.0;
      BLD   103;
      A     I    302.6;
      =     L      0.1;
      BLD   103;
      A     I    302.7;
      =     L      0.2;
      BLD   103;
      A     I    303.0;
      =     L      0.3;
      BLD   103;
      A     I    303.1;
      =     L      0.4;
      BLD   103;
      A     I    303.2;
      =     L      0.5;
      BLD   103;
      A     I    303.3;
      =     L      0.6;
      BLD   103;
      A     I    303.4;
      =     L      0.7;
      BLD   103;
      A     I    303.5;
      =     L      1.0;
      BLD   103;
      A     I    304.0;
      =     L      1.1;
      BLD   103;
      A     I    304.1;
      =     L      1.2;
      BLD   103;
      A     M    740.2;
      =     L      2.1;
      BLD   103;
      A     M    740.3;
      =     L      2.2;
      BLD   103;
      AN    M    504.0;
      AN    M    504.1;
      AN    M   6060.0;
      AN    M   6260.0;
      AN    M   6280.0;
      AN    M    504.2;
      A     M    500.2;
      =     L      2.3;
      BLD   103;
      A(    ;
      O     I      0.1;
      O     M   4120.1;
      )     ;
      =     L      2.5;
      BLD   103;
      A     M      0.5;
      =     L      2.6;
      BLD   103;
      CALL #S705_TL_DC_LATCH1 (
           Enable_Aux               := L      0.0,
           Adv_Amount               := 5,
           Ret_Amount               := 5,
           LS_Adv1                  := L      0.1,
           LS_Ret1                  := L      0.2,
           LS_Adv2                  := L      0.3,
           LS_Ret2                  := L      0.4,
           LS_Adv3                  := L      0.5,
           LS_Ret3                  := L      0.6,
           LS_Adv4                  := L      0.7,
           LS_Ret4                  := L      1.0,
           LS_Adv5                  := L      1.1,
           LS_Ret5                  := L      1.2,
           SOL_Adv                  := L      2.1,
           SOL_Ret                  := L      2.2,
           M_Ready                  := L      2.3,
           T_CHK1                   := T#4S,
           T_CHK2                   := T#4S,
           PB_Error_Rst             := L      2.5,
           M_FLICK                  := L      2.6,
           M_Adv_Err                := M    750.2,
           M_Ret_Err                := M    750.3,
           Visu_Adv                 := DB51.DBW  124,
           Visu_Ret                 := DB51.DBW  126);
      NOP   0;
NETWORK
TITLE =
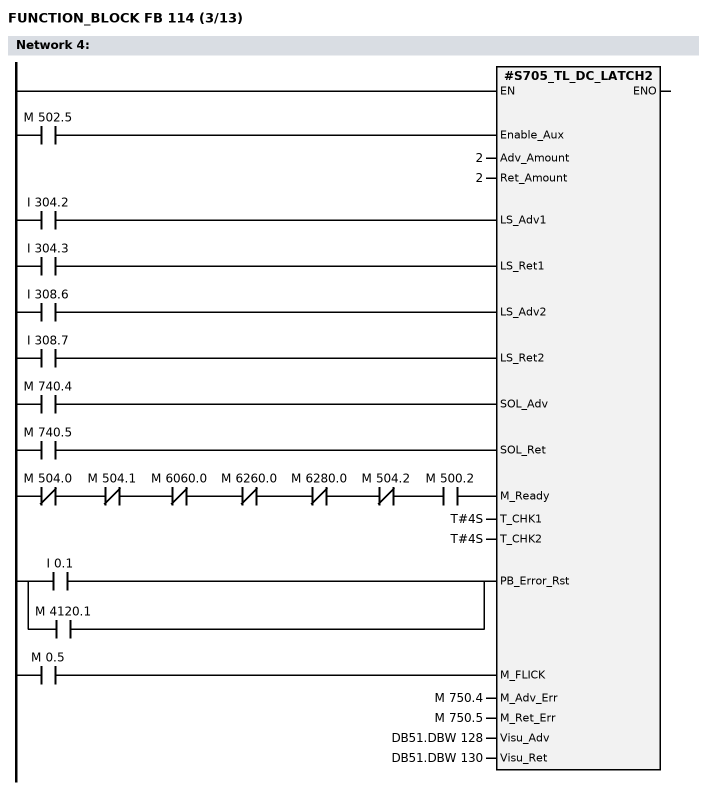

      A     M    502.5;
      =     L      0.0;
      BLD   103;
      A     I    304.2;
      =     L      0.1;
      BLD   103;
      A     I    304.3;
      =     L      0.2;
      BLD   103;
      A     I    308.6;
      =     L      0.3;
      BLD   103;
      A     I    308.7;
      =     L      0.4;
      BLD   103;
      A     M    740.4;
      =     L      2.1;
      BLD   103;
      A     M    740.5;
      =     L      2.2;
      BLD   103;
      AN    M    504.0;
      AN    M    504.1;
      AN    M   6060.0;
      AN    M   6260.0;
      AN    M   6280.0;
      AN    M    504.2;
      A     M    500.2;
      =     L      2.3;
      BLD   103;
      A(    ;
      O     I      0.1;
      O     M   4120.1;
      )     ;
      =     L      2.5;
      BLD   103;
      A     M      0.5;
      =     L      2.6;
      BLD   103;
      CALL #S705_TL_DC_LATCH2 (
           Enable_Aux               := L      0.0,
           Adv_Amount               := 2,
           Ret_Amount               := 2,
           LS_Adv1                  := L      0.1,
           LS_Ret1                  := L      0.2,
           LS_Adv2                  := L      0.3,
           LS_Ret2                  := L      0.4,
           SOL_Adv                  := L      2.1,
           SOL_Ret                  := L      2.2,
           M_Ready                  := L      2.3,
           T_CHK1                   := T#4S,
           T_CHK2                   := T#4S,
           PB_Error_Rst             := L      2.5,
           M_FLICK                  := L      2.6,
           M_Adv_Err                := M    750.4,
           M_Ret_Err                := M    750.5,
           Visu_Adv                 := DB51.DBW  128,
           Visu_Ret                 := DB51.DBW  130);
      NOP   0;
NETWORK
TITLE =
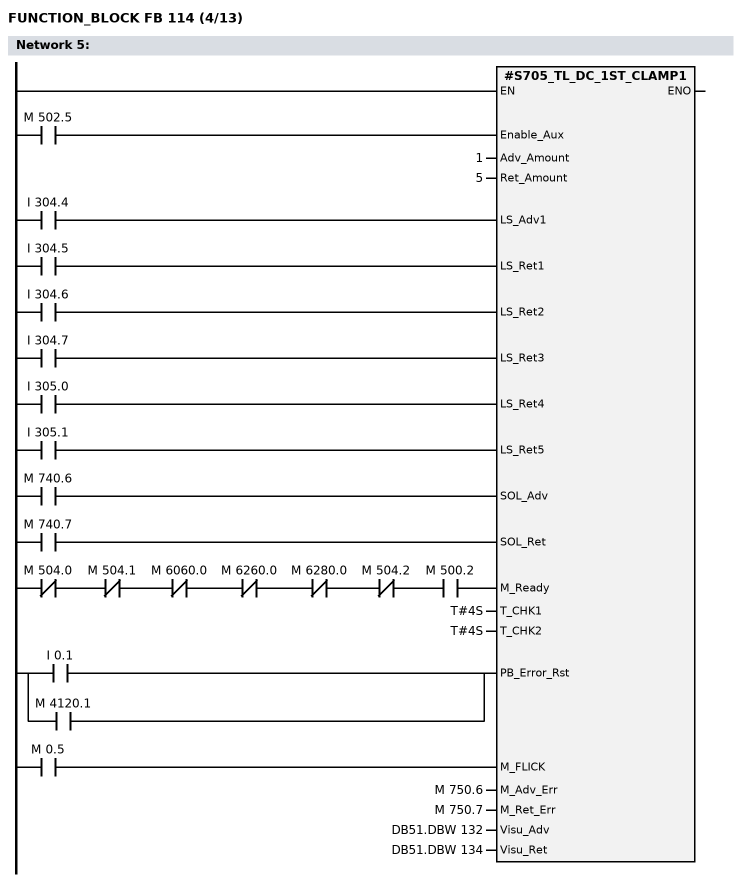

